LIN {X 0,Y 256.443,Z 273.526,A -85,B 0,C 180,E1 -18716.858,E2 -18716.858} C_VEL
LIN {X 0,Y 256.695,Z 273.51,A -85,B 0,C 180,E1 -18718.431,E2 -18718.431} C_VEL
LIN {X 0,Y 256.584,Z 273.506,A -85,B 0,C 180,E1 -18722.128,E2 -18722.128} C_VEL
LIN {X 0,Y 255.761,Z 273.619,A -85,B 0,C 180,E1 -18723.437,E2 -18723.437} C_VEL
LIN {X 0,Y 252.839,Z 273.986,A -85,B 0,C 180,E1 -18725.572,E2 -18725.572} C_VEL
LIN {X 0,Y 250.455,Z 274.274,A -85,B 0,C 180,E1 -18727.309,E2 -18727.309} C_VEL
LIN {X 0,Y 249.449,Z 274.4,A -85,B 0,C 180,E1 -18728.656,E2 -18728.656} C_VEL
LIN {X 0,Y 249.37,Z 274.413,A -85,B 0,C 180,E1 -18729.112,E2 -18729.112} C_VEL
LIN {X 0,Y 249.184,Z 274.428,A -85,B 0,C 180,E1 -18733.04,E2 -18733.04} C_VEL
LIN {X 0,Y 249.193,Z 274.444,A -85,B 0,C 180,E1 -18736.486,E2 -18736.486} C_VEL
LIN {X 0,Y 249.077,Z 274.451,A -85,B 0,C 180,E1 -18741.519,E2 -18741.519} C_VEL
LIN {X 0,Y 249.078,Z 274.447,A -85,B 0,C 180,E1 -18745.457,E2 -18745.457} C_VEL
LIN {X 0,Y 249.021,Z 274.443,A -85,B 0,C 180,E1 -18748.968,E2 -18748.968} C_VEL
LIN {X 0,Y 249.023,Z 274.449,A -85,B 0,C 180,E1 -18752.427,E2 -18752.427} C_VEL
LIN {X 0,Y 249.029,Z 274.467,A -85,B 0,C 180,E1 -18756.345,E2 -18756.345} C_VEL
LIN {X 0,Y 248.977,Z 274.467,A -85,B 0,C 180,E1 -18760.484,E2 -18760.484} C_VEL
LIN {X 0,Y 249.005,Z 274.668,A -85,B 0,C 180,E1 -18763.299,E2 -18763.299} C_VEL
LIN {X 0,Y 251.939,Z 284.13,A -85,B 0,C 180,E1 -18767.093,E2 -18767.093} C_VEL
LIN {X 0,Y 254.692,Z 293.785,A -85,B 0,C 180,E1 -18770.605,E2 -18770.605} C_VEL
LIN {X 0,Y 256.851,Z 302.565,A -85,B 0,C 180,E1 -18773.556,E2 -18773.556} C_VEL
LIN {X 0,Y 257.592,Z 305.745,A -85,B 0,C 180,E1 -18774.479,E2 -18774.479} C_VEL
LIN {X 0,Y 262.27,Z 316.515,A -85,B 0,C 180,E1 -18775.675,E2 -18775.675} C_VEL
LIN {X 0,Y 263.173,Z 319.74,A -85,B 0,C 180,E1 -18775.93,E2 -18775.93} C_VEL
LIN {X 0,Y 267.638,Z 349.75,A -85,B 0,C 180,E1 -18777.608,E2 -18777.608} C_VEL
LIN {X 0,Y 270.306,Z 373.324,A -85,B 0,C 180,E1 -18778.747,E2 -18778.747} C_VEL
LIN {X 0,Y 270.85,Z 381.222,A -85,B 0,C 180,E1 -18779.071,E2 -18779.071} C_VEL
LIN {X 0,Y 269.246,Z 418.517,A -85,B 0,C 180,E1 -18780.065,E2 -18780.065} C_VEL
LIN {X 0,Y 267.955,Z 432.124,A -85,B 0,C 180,E1 -18780.704,E2 -18780.704} C_VEL
LIN {X 0,Y 266.124,Z 445.126,A -85,B 0,C 180,E1 -18781.617,E2 -18781.617} C_VEL
LIN {X 0,Y 263.547,Z 457.746,A -85,B 0,C 180,E1 -18782.827,E2 -18782.827} C_VEL
LIN {X 0,Y 260.85,Z 469.017,A -85,B 0,C 180,E1 -18784.25,E2 -18784.25} C_VEL
LIN {X 0,Y 258.114,Z 479.21,A -85,B 0,C 180,E1 -18785.894,E2 -18785.894} C_VEL
LIN {X 0,Y 255.483,Z 488.439,A -85,B 0,C 180,E1 -18787.775,E2 -18787.775} C_VEL
LIN {X 0,Y 252.796,Z 497.481,A -85,B 0,C 180,E1 -18790.089,E2 -18790.089} C_VEL
LIN {X 0,Y 250.941,Z 504.121,A -85,B 0,C 180,E1 -18792.218,E2 -18792.218} C_VEL
LIN {X 0,Y 249.474,Z 509.836,A -85,B 0,C 180,E1 -18794.477,E2 -18794.477} C_VEL
LIN {X 0,Y 248.297,Z 514.754,A -85,B 0,C 180,E1 -18796.912,E2 -18796.912} C_VEL
LIN {X 0,Y 247.635,Z 518.587,A -85,B 0,C 180,E1 -18799.369,E2 -18799.369} C_VEL
LIN {X 0,Y 247.49,Z 521.437,A -85,B 0,C 180,E1 -18801.837,E2 -18801.837} C_VEL
LIN {X 0,Y 247.65,Z 522.833,A -85,B 0,C 180,E1 -18803.481,E2 -18803.481} C_VEL
LIN {X 0,Y 247.793,Z 523.809,A -85,B 0,C 180,E1 -18805.118,E2 -18805.118} C_VEL
LIN {X 0,Y 248.089,Z 524.353,A -85,B 0,C 180,E1 -18806.751,E2 -18806.751} C_VEL
LIN {X 0,Y 248.279,Z 524.479,A -85,B 0,C 180,E1 -18808.377,E2 -18808.377} C_VEL
LIN {X 0,Y 248.404,Z 524.194,A -85,B 0,C 180,E1 -18809.999,E2 -18809.999} C_VEL
LIN {X 0,Y 248.339,Z 523.474,A -85,B 0,C 180,E1 -18811.621,E2 -18811.621} C_VEL
LIN {X 0,Y 248.24,Z 522.282,A -85,B 0,C 180,E1 -18813.245,E2 -18813.245} C_VEL
LIN {X 0,Y 247.888,Z 519.656,A -85,B 0,C 180,E1 -18815.694,E2 -18815.694} C_VEL
LIN {X 0,Y 247.682,Z 515.965,A -85,B 0,C 180,E1 -18818.156,E2 -18818.156} C_VEL
LIN {X 0,Y 247.779,Z 511.131,A -85,B 0,C 180,E1 -18820.623,E2 -18820.623} C_VEL
LIN {X 0,Y 248.462,Z 503.88,A -85,B 0,C 180,E1 -18823.494,E2 -18823.494} C_VEL
LIN {X 0,Y 249.454,Z 496.031,A -85,B 0,C 180,E1 -18825.943,E2 -18825.943} C_VEL
LIN {X 0,Y 250.831,Z 488.044,A -85,B 0,C 180,E1 -18827.95,E2 -18827.95} C_VEL
LIN {X 0,Y 252.264,Z 479.373,A -85,B 0,C 180,E1 -18829.742,E2 -18829.742} C_VEL
LIN {X 0,Y 254.056,Z 468.801,A -85,B 0,C 180,E1 -18831.501,E2 -18831.501} C_VEL
LIN {X 0,Y 255.949,Z 457.085,A -85,B 0,C 180,E1 -18833.033,E2 -18833.033} C_VEL
LIN {X 0,Y 257.624,Z 444.652,A -85,B 0,C 180,E1 -18834.26,E2 -18834.26} C_VEL
LIN {X 0,Y 258.91,Z 431.527,A -85,B 0,C 180,E1 -18835.202,E2 -18835.202} C_VEL
LIN {X 0,Y 259.783,Z 418.703,A -85,B 0,C 180,E1 -18835.809,E2 -18835.809} C_VEL
LIN {X 0,Y 260.834,Z 377.068,A -85,B 0,C 180,E1 -18836.957,E2 -18836.957} C_VEL
LIN {X 0,Y 257.271,Z 335.818,A -85,B 0,C 180,E1 -18838.516,E2 -18838.516} C_VEL
LIN {X 0,Y 254.216,Z 308.569,A -85,B 0,C 180,E1 -18839.693,E2 -18839.693} C_VEL
LIN {X 0,Y 254.746,Z 304.307,A -85,B 0,C 180,E1 -18840.668,E2 -18840.668} C_VEL
LIN {X 0,Y 254.864,Z 300.787,A -85,B 0,C 180,E1 -18841.595,E2 -18841.595} C_VEL
LIN {X 0,Y 252.702,Z 289.84,A -85,B 0,C 180,E1 -18844.757,E2 -18844.757} C_VEL
LIN {X 0,Y 250.099,Z 278.579,A -85,B 0,C 180,E1 -18848.184,E2 -18848.184} C_VEL
LIN {X 0,Y 249.018,Z 274.551,A -85,B 0,C 180,E1 -18849.55,E2 -18849.55} C_VEL
LIN {X 0,Y 248.978,Z 274.464,A -85,B 0,C 180,E1 -18852.785,E2 -18852.785} C_VEL
LIN {X 0,Y 248.973,Z 274.461,A -85,B 0,C 180,E1 -18857.354,E2 -18857.354} C_VEL
LIN {X 0,Y 249.033,Z 274.456,A -85,B 0,C 180,E1 -18862.201,E2 -18862.201} C_VEL
LIN {X 0,Y 249.036,Z 274.459,A -85,B 0,C 180,E1 -18865.638,E2 -18865.638} C_VEL
LIN {X 0,Y 248.987,Z 274.465,A -85,B 0,C 180,E1 -18869.464,E2 -18869.464} C_VEL
LIN {X 0,Y 249.021,Z 274.459,A -85,B 0,C 180,E1 -18873.156,E2 -18873.156} C_VEL
LIN {X 0,Y 249.043,Z 274.459,A -85,B 0,C 180,E1 -18876.729,E2 -18876.729} C_VEL
LIN {X 0,Y 249.039,Z 274.46,A -85,B 0,C 180,E1 -18880.206,E2 -18880.206} C_VEL
LIN {X 0,Y 249.149,Z 274.443,A -85,B 0,C 180,E1 -18883.616,E2 -18883.616} C_VEL
LIN {X 0,Y 249.224,Z 274.431,A -85,B 0,C 180,E1 -18888.616,E2 -18888.616} C_VEL
LIN {X 0,Y 249.408,Z 274.407,A -85,B 0,C 180,E1 -18891.901,E2 -18891.901} C_VEL
LIN {X 0,Y 249.253,Z 274.436,A -85,B 0,C 180,E1 -18895.148,E2 -18895.148} C_VEL
LIN {X 0,Y 249.648,Z 274.372,A -85,B 0,C 180,E1 -18898.387,E2 -18898.387} C_VEL
LIN {X 0,Y 249.647,Z 274.381,A -85,B 0,C 180,E1 -18901.614,E2 -18901.614} C_VEL
LIN {X 0,Y 249.398,Z 274.408,A -85,B 0,C 180,E1 -18906.665,E2 -18906.665} C_VEL
LIN {X 0,Y 249.324,Z 274.413,A -85,B 0,C 180,E1 -18909.738,E2 -18909.738} C_VEL
LIN {X 0,Y 249.163,Z 274.443,A -85,B 0,C 180,E1 -18914.706,E2 -18914.706} C_VEL
LIN {X 0,Y 249.087,Z 274.44,A -85,B 0,C 180,E1 -18918.082,E2 -18918.082} C_VEL
LIN {X 0,Y 249.036,Z 274.462,A -85,B 0,C 180,E1 -18921.523,E2 -18921.523} C_VEL
LIN {X 0,Y 249.037,Z 274.45,A -85,B 0,C 180,E1 -18925.441,E2 -18925.441} C_VEL
LIN {X 0,Y 249.017,Z 274.464,A -85,B 0,C 180,E1 -18928.969,E2 -18928.969} C_VEL
LIN {X 0,Y 249.02,Z 274.456,A -85,B 0,C 180,E1 -18932.428,E2 -18932.428} C_VEL
LIN {X 0,Y 249.008,Z 274.468,A -85,B 0,C 180,E1 -18936.35,E2 -18936.35} C_VEL
LIN {X 0,Y 248.974,Z 274.454,A -85,B 0,C 180,E1 -18940.485,E2 -18940.485} C_VEL
LIN {X 0,Y 248.958,Z 274.447,A -85,B 0,C 180,E1 -18944.89,E2 -18944.89} C_VEL
LIN {X 0,Y 248.976,Z 274.469,A -85,B 0,C 180,E1 -18947.356,E2 -18947.356} C_VEL
LIN {X 0,Y 249.041,Z 274.433,A -85,B 0,C 180,E1 -18952.202,E2 -18952.202} C_VEL
LIN {X 0,Y 249.041,Z 274.46,A -85,B 0,C 180,E1 -18955.641,E2 -18955.641} C_VEL
LIN {X 0,Y 248.992,Z 274.45,A -85,B 0,C 180,E1 -18959.467,E2 -18959.467} C_VEL
LIN {X 0,Y 249.013,Z 274.466,A -85,B 0,C 180,E1 -18963.157,E2 -18963.157} C_VEL
LIN {X 0,Y 249.007,Z 274.466,A -85,B 0,C 180,E1 -18966.727,E2 -18966.727} C_VEL
LIN {X 0,Y 249.069,Z 274.697,A -85,B 0,C 180,E1 -18968.264,E2 -18968.264} C_VEL
LIN {X 0,Y 249.342,Z 275.779,A -85,B 0,C 180,E1 -18968.528,E2 -18968.528} C_VEL
LIN {X 0,Y 256.786,Z 291.191,A -85,B 0,C 180,E1 -18969.864,E2 -18969.864} C_VEL
LIN {X 0,Y 262.664,Z 305.025,A -85,B 0,C 180,E1 -18970.889,E2 -18970.889} C_VEL
LIN {X 0,Y 261.449,Z 360.767,A -85,B 0,C 180,E1 -18972.438,E2 -18972.438} C_VEL
LIN {X 0,Y 260.873,Z 373.588,A -85,B 0,C 180,E1 -18973.066,E2 -18973.066} C_VEL
LIN {X 0,Y 260.178,Z 386.354,A -85,B 0,C 180,E1 -18974.028,E2 -18974.028} C_VEL
LIN {X 0,Y 258.96,Z 398.602,A -85,B 0,C 180,E1 -18975.261,E2 -18975.261} C_VEL
LIN {X 0,Y 257.48,Z 410.104,A -85,B 0,C 180,E1 -18976.786,E2 -18976.786} C_VEL
LIN {X 0,Y 256.054,Z 420.419,A -85,B 0,C 180,E1 -18978.523,E2 -18978.523} C_VEL
LIN {X 0,Y 254.596,Z 429.735,A -85,B 0,C 180,E1 -18980.467,E2 -18980.467} C_VEL
LIN {X 0,Y 252.927,Z 438.733,A -85,B 0,C 180,E1 -18982.818,E2 -18982.818} C_VEL
LIN {X 0,Y 251.555,Z 445.985,A -85,B 0,C 180,E1 -18985.193,E2 -18985.193} C_VEL
LIN {X 0,Y 250.513,Z 451.8,A -85,B 0,C 180,E1 -18987.589,E2 -18987.589} C_VEL
LIN {X 0,Y 249.731,Z 456.398,A -85,B 0,C 180,E1 -18990.001,E2 -18990.001} C_VEL
LIN {X 0,Y 249.118,Z 459.929,A -85,B 0,C 180,E1 -18992.426,E2 -18992.426} C_VEL
LIN {X 0,Y 248.925,Z 462.45,A -85,B 0,C 180,E1 -18994.859,E2 -18994.859} C_VEL
LIN {X 0,Y 248.891,Z 463.645,A -85,B 0,C 180,E1 -18996.486,E2 -18996.486} C_VEL
LIN {X 0,Y 249.017,Z 464.801,A -85,B 0,C 180,E1 -18999.75,E2 -18999.75} C_VEL
LIN {X 0,Y 249.606,Z 464.433,A -85,B 0,C 180,E1 -19003.018,E2 -19003.018} C_VEL
LIN {X 0,Y 250.697,Z 462.408,A -85,B 0,C 180,E1 -19006.281,E2 -19006.281} C_VEL
LIN {X 0,Y 251.679,Z 460.33,A -85,B 0,C 180,E1 -19008.297,E2 -19008.297} C_VEL
LIN {X 0,Y 253.326,Z 456.162,A -85,B 0,C 180,E1 -19011.141,E2 -19011.141} C_VEL
LIN {X 0,Y 255.106,Z 451.378,A -85,B 0,C 180,E1 -19013.545,E2 -19013.545} C_VEL
LIN {X 0,Y 257.245,Z 445.293,A -85,B 0,C 180,E1 -19015.921,E2 -19015.921} C_VEL
LIN {X 0,Y 259.642,Z 437.642,A -85,B 0,C 180,E1 -19018.274,E2 -19018.274} C_VEL
LIN {X 0,Y 261.926,Z 429.739,A -85,B 0,C 180,E1 -19020.205,E2 -19020.205} C_VEL
LIN {X 0,Y 264.26,Z 420.034,A -85,B 0,C 180,E1 -19022.134,E2 -19022.134} C_VEL
LIN {X 0,Y 266.613,Z 409.146,A -85,B 0,C 180,E1 -19023.839,E2 -19023.839} C_VEL
LIN {X 0,Y 268.486,Z 398.379,A -85,B 0,C 180,E1 -19025.161,E2 -19025.161} C_VEL
LIN {X 0,Y 269.94,Z 387.778,A -85,B 0,C 180,E1 -19026.186,E2 -19026.186} C_VEL
LIN {X 0,Y 271.093,Z 375.462,A -85,B 0,C 180,E1 -19027.088,E2 -19027.088} C_VEL
LIN {X 0,Y 271.773,Z 363.252,A -85,B 0,C 180,E1 -19027.707,E2 -19027.707} C_VEL
LIN {X 0,Y 272.781,Z 328.656,A -85,B 0,C 180,E1 -19028.694,E2 -19028.694} C_VEL
LIN {X 0,Y 273.176,Z 316.973,A -85,B 0,C 180,E1 -19029.004,E2 -19029.004} C_VEL
LIN {X 0,Y 265.765,Z 302.535,A -85,B 0,C 180,E1 -19030.616,E2 -19030.616} C_VEL
LIN {X 0,Y 258.181,Z 289.71,A -85,B 0,C 180,E1 -19032.334,E2 -19032.334} C_VEL
LIN {X 0,Y 253.23,Z 282.015,A -85,B 0,C 180,E1 -19033.51,E2 -19033.51} C_VEL
LIN {X 0,Y 251.177,Z 278.766,A -85,B 0,C 180,E1 -19034.02,E2 -19034.02} C_VEL
LIN {X 0,Y 249.479,Z 276.328,A -85,B 0,C 180,E1 -19034.45,E2 -19034.45} C_VEL
LIN {X 0,Y 249.065,Z 275,A -85,B 0,C 180,E1 -19034.691,E2 -19034.691} C_VEL
LIN {X 0,Y 248.967,Z 274.504,A -85,B 0,C 180,E1 -19035.112,E2 -19035.112} C_VEL
LIN {X 0,Y 248.979,Z 274.473,A -85,B 0,C 180,E1 -19039.516,E2 -19039.516} C_VEL
LIN {X 0,Y 249.012,Z 274.438,A -85,B 0,C 180,E1 -19043.651,E2 -19043.651} C_VEL
LIN {X 0,Y 249.03,Z 274.435,A -85,B 0,C 180,E1 -19047.848,E2 -19047.848} C_VEL
LIN {X 0,Y 249.038,Z 274.432,A -85,B 0,C 180,E1 -19051.33,E2 -19051.33} C_VEL
LIN {X 0,Y 249.1,Z 274.444,A -85,B 0,C 180,E1 -19054.962,E2 -19054.962} C_VEL
LIN {X 0,Y 249.089,Z 274.4,A -85,B 0,C 180,E1 -19058.604,E2 -19058.604} C_VEL
LIN {X 0,Y 249.241,Z 274.436,A -85,B 0,C 180,E1 -19063.621,E2 -19063.621} C_VEL
LIN {X 0,Y 249.24,Z 274.437,A -85,B 0,C 180,E1 -19068.616,E2 -19068.616} C_VEL
LIN {X 0,Y 249.414,Z 274.405,A -85,B 0,C 180,E1 -19071.9,E2 -19071.9} C_VEL
LIN {X 0,Y 249.253,Z 274.424,A -85,B 0,C 180,E1 -19075.147,E2 -19075.147} C_VEL
LIN {X 0,Y 249.655,Z 274.387,A -85,B 0,C 180,E1 -19078.386,E2 -19078.386} C_VEL
LIN {X 0,Y 249.561,Z 274.381,A -85,B 0,C 180,E1 -19082.058,E2 -19082.058} C_VEL
LIN {X 0,Y 249.421,Z 274.403,A -85,B 0,C 180,E1 -19086.471,E2 -19086.471} C_VEL
LIN {X 0,Y 249.37,Z 274.413,A -85,B 0,C 180,E1 -19089.112,E2 -19089.112} C_VEL
LIN {X 0,Y 248.682,Z 274.51,A -85,B 0,C 180,E1 -19090.458,E2 -19090.458} C_VEL
LIN {X 0,Y 245.733,Z 274.877,A -85,B 0,C 180,E1 -19092.65,E2 -19092.65} C_VEL
LIN {X 0,Y 243.238,Z 275.182,A -85,B 0,C 180,E1 -19094.436,E2 -19094.436} C_VEL
LIN {X 0,Y 242.186,Z 275.318,A -85,B 0,C 180,E1 -19095.824,E2 -19095.824} C_VEL
LIN {X 0,Y 242.111,Z 275.322,A -85,B 0,C 180,E1 -19096.295,E2 -19096.295} C_VEL
LIN {X 0,Y 242.021,Z 275.339,A -85,B 0,C 180,E1 -19100.393,E2 -19100.393} C_VEL
LIN {X 0,Y 242.021,Z 275.34,A -85,B 0,C 180,E1 -19103.988,E2 -19103.988} C_VEL
LIN {X 0,Y 241.953,Z 275.313,A -85,B 0,C 180,E1 -19107.694,E2 -19107.694} C_VEL
LIN {X 0,Y 241.946,Z 275.344,A -85,B 0,C 180,E1 -19111.524,E2 -19111.524} C_VEL
LIN {X 0,Y 242.004,Z 275.33,A -85,B 0,C 180,E1 -19115.597,E2 -19115.597} C_VEL
LIN {X 0,Y 241.938,Z 275.334,A -85,B 0,C 180,E1 -19119.722,E2 -19119.722} C_VEL
LIN {X 0,Y 241.957,Z 275.593,A -85,B 0,C 180,E1 -19122.09,E2 -19122.09} C_VEL
LIN {X 0,Y 244.787,Z 284.528,A -85,B 0,C 180,E1 -19125.87,E2 -19125.87} C_VEL
LIN {X 0,Y 247.628,Z 294.176,A -85,B 0,C 180,E1 -19129.57,E2 -19129.57} C_VEL
LIN {X 0,Y 250.128,Z 304.192,A -85,B 0,C 180,E1 -19133.037,E2 -19133.037} C_VEL
LIN {X 0,Y 254.27,Z 313.334,A -85,B 0,C 180,E1 -19134.196,E2 -19134.196} C_VEL
LIN {X 0,Y 257.472,Z 320.978,A -85,B 0,C 180,E1 -19135.025,E2 -19135.025} C_VEL
LIN {X 0,Y 261.882,Z 351.317,A -85,B 0,C 180,E1 -19136.777,E2 -19136.777} C_VEL
LIN {X 0,Y 264.447,Z 374.596,A -85,B 0,C 180,E1 -19137.935,E2 -19137.935} C_VEL
LIN {X 0,Y 264.899,Z 382.546,A -85,B 0,C 180,E1 -19138.26,E2 -19138.26} C_VEL
LIN {X 0,Y 263.417,Z 416.986,A -85,B 0,C 180,E1 -19139.194,E2 -19139.194} C_VEL
LIN {X 0,Y 262.11,Z 430.421,A -85,B 0,C 180,E1 -19139.818,E2 -19139.818} C_VEL
LIN {X 0,Y 260.286,Z 443.122,A -85,B 0,C 180,E1 -19140.699,E2 -19140.699} C_VEL
LIN {X 0,Y 258.002,Z 454.457,A -85,B 0,C 180,E1 -19141.751,E2 -19141.751} C_VEL
LIN {X 0,Y 255.108,Z 466.171,A -85,B 0,C 180,E1 -19143.185,E2 -19143.185} C_VEL
LIN {X 0,Y 252.217,Z 476.733,A -85,B 0,C 180,E1 -19144.853,E2 -19144.853} C_VEL
LIN {X 0,Y 249.424,Z 486.3,A -85,B 0,C 180,E1 -19146.767,E2 -19146.767} C_VEL
LIN {X 0,Y 246.544,Z 495.562,A -85,B 0,C 180,E1 -19149.125,E2 -19149.125} C_VEL
LIN {X 0,Y 244.287,Z 503.086,A -85,B 0,C 180,E1 -19151.551,E2 -19151.551} C_VEL
LIN {X 0,Y 242.606,Z 509.188,A -85,B 0,C 180,E1 -19154.025,E2 -19154.025} C_VEL
LIN {X 0,Y 241.348,Z 514.06,A -85,B 0,C 180,E1 -19156.528,E2 -19156.528} C_VEL
LIN {X 0,Y 240.602,Z 517.848,A -85,B 0,C 180,E1 -19159.055,E2 -19159.055} C_VEL
LIN {X 0,Y 240.403,Z 520.657,A -85,B 0,C 180,E1 -19161.594,E2 -19161.594} C_VEL
LIN {X 0,Y 240.57,Z 522.085,A -85,B 0,C 180,E1 -19163.352,E2 -19163.352} C_VEL
LIN {X 0,Y 241.011,Z 523.508,A -85,B 0,C 180,E1 -19166.656,E2 -19166.656} C_VEL
LIN {X 0,Y 241.227,Z 523.62,A -85,B 0,C 180,E1 -19168.33,E2 -19168.33} C_VEL
LIN {X 0,Y 241.355,Z 523.318,A -85,B 0,C 180,E1 -19169.999,E2 -19169.999} C_VEL
LIN {X 0,Y 241.29,Z 522.569,A -85,B 0,C 180,E1 -19171.668,E2 -19171.668} C_VEL
LIN {X 0,Y 241.157,Z 521.345,A -85,B 0,C 180,E1 -19173.341,E2 -19173.341} C_VEL
LIN {X 0,Y 240.816,Z 518.678,A -85,B 0,C 180,E1 -19175.862,E2 -19175.862} C_VEL
LIN {X 0,Y 240.605,Z 514.94,A -85,B 0,C 180,E1 -19178.397,E2 -19178.397} C_VEL
LIN {X 0,Y 240.75,Z 510.06,A -85,B 0,C 180,E1 -19180.937,E2 -19180.937} C_VEL
LIN {X 0,Y 241.494,Z 502.756,A -85,B 0,C 180,E1 -19183.891,E2 -19183.891} C_VEL
LIN {X 0,Y 242.52,Z 494.817,A -85,B 0,C 180,E1 -19186.411,E2 -19186.411} C_VEL
LIN {X 0,Y 243.992,Z 486.755,A -85,B 0,C 180,E1 -19188.471,E2 -19188.471} C_VEL
LIN {X 0,Y 245.779,Z 476.927,A -85,B 0,C 180,E1 -19190.504,E2 -19190.504} C_VEL
LIN {X 0,Y 247.572,Z 466.003,A -85,B 0,C 180,E1 -19192.313,E2 -19192.313} C_VEL
LIN {X 0,Y 249.139,Z 457.076,A -85,B 0,C 180,E1 -19193.48,E2 -19193.48} C_VEL
LIN {X 0,Y 250.862,Z 444.998,A -85,B 0,C 180,E1 -19194.737,E2 -19194.737} C_VEL
LIN {X 0,Y 252.189,Z 432.293,A -85,B 0,C 180,E1 -19195.701,E2 -19195.701} C_VEL
LIN {X 0,Y 253.157,Z 419.171,A -85,B 0,C 180,E1 -19196.37,E2 -19196.37} C_VEL
LIN {X 0,Y 254.296,Z 377.496,A -85,B 0,C 180,E1 -19197.563,E2 -19197.563} C_VEL
LIN {X 0,Y 250.733,Z 335.752,A -85,B 0,C 180,E1 -19199.195,E2 -19199.195} C_VEL
LIN {X 0,Y 247.598,Z 307.785,A -85,B 0,C 180,E1 -19200.449,E2 -19200.449} C_VEL
LIN {X 0,Y 247.883,Z 305.078,A -85,B 0,C 180,E1 -19201.028,E2 -19201.028} C_VEL
LIN {X 0,Y 247.794,Z 301.329,A -85,B 0,C 180,E1 -19202.064,E2 -19202.064} C_VEL
LIN {X 0,Y 245.385,Z 289.262,A -85,B 0,C 180,E1 -19205.681,E2 -19205.681} C_VEL
LIN {X 0,Y 243.108,Z 279.773,A -85,B 0,C 180,E1 -19208.69,E2 -19208.69} C_VEL
LIN {X 0,Y 241.969,Z 275.448,A -85,B 0,C 180,E1 -19210.189,E2 -19210.189} C_VEL
LIN {X 0,Y 241.894,Z 275.323,A -85,B 0,C 180,E1 -19214.208,E2 -19214.208} C_VEL
LIN {X 0,Y 241.902,Z 275.351,A -85,B 0,C 180,E1 -19218.07,E2 -19218.07} C_VEL
LIN {X 0,Y 241.978,Z 275.335,A -85,B 0,C 180,E1 -19222.416,E2 -19222.416} C_VEL
LIN {X 0,Y 241.971,Z 275.333,A -85,B 0,C 180,E1 -19226.506,E2 -19226.506} C_VEL
LIN {X 0,Y 241.964,Z 275.343,A -85,B 0,C 180,E1 -19230.614,E2 -19230.614} C_VEL
LIN {X 0,Y 242.025,Z 275.326,A -85,B 0,C 180,E1 -19234.178,E2 -19234.178} C_VEL
LIN {X 0,Y 241.984,Z 275.342,A -85,B 0,C 180,E1 -19238.334,E2 -19238.334} C_VEL
LIN {X 0,Y 242.105,Z 275.317,A -85,B 0,C 180,E1 -19243.318,E2 -19243.318} C_VEL
LIN {X 0,Y 242.158,Z 275.315,A -85,B 0,C 180,E1 -19248.279,E2 -19248.279} C_VEL
LIN {X 0,Y 242.362,Z 275.284,A -85,B 0,C 180,E1 -19251.664,E2 -19251.664} C_VEL
LIN {X 0,Y 242.386,Z 275.29,A -85,B 0,C 180,E1 -19253.34,E2 -19253.34} C_VEL
LIN {X 0,Y 242.608,Z 275.248,A -85,B 0,C 180,E1 -19258.34,E2 -19258.34} C_VEL
LIN {X 0,Y 242.606,Z 275.258,A -85,B 0,C 180,E1 -19261.66,E2 -19261.66} C_VEL
LIN {X 0,Y 242.38,Z 275.282,A -85,B 0,C 180,E1 -19266.661,E2 -19266.661} C_VEL
LIN {X 0,Y 242.252,Z 275.294,A -85,B 0,C 180,E1 -19270.025,E2 -19270.025} C_VEL
LIN {X 0,Y 242.113,Z 275.319,A -85,B 0,C 180,E1 -19275.145,E2 -19275.145} C_VEL
LIN {X 0,Y 242.023,Z 275.323,A -85,B 0,C 180,E1 -19278.629,E2 -19278.629} C_VEL
LIN {X 0,Y 241.966,Z 275.345,A -85,B 0,C 180,E1 -19282.185,E2 -19282.185} C_VEL
LIN {X 0,Y 241.98,Z 275.327,A -85,B 0,C 180,E1 -19285.828,E2 -19285.828} C_VEL
LIN {X 0,Y 241.956,Z 275.345,A -85,B 0,C 180,E1 -19289.591,E2 -19289.591} C_VEL
LIN {X 0,Y 241.973,Z 275.33,A -85,B 0,C 180,E1 -19293.494,E2 -19293.494} C_VEL
LIN {X 0,Y 241.979,Z 275.344,A -85,B 0,C 180,E1 -19297.585,E2 -19297.585} C_VEL
LIN {X 0,Y 241.896,Z 275.314,A -85,B 0,C 180,E1 -19301.932,E2 -19301.932} C_VEL
LIN {X 0,Y 241.897,Z 275.347,A -85,B 0,C 180,E1 -19306.582,E2 -19306.582} C_VEL
LIN {X 0,Y 241.991,Z 275.314,A -85,B 0,C 180,E1 -19311.643,E2 -19311.643} C_VEL
LIN {X 0,Y 241.972,Z 275.324,A -85,B 0,C 180,E1 -19314.488,E2 -19314.488} C_VEL
LIN {X 0,Y 241.947,Z 275.334,A -85,B 0,C 180,E1 -19318.477,E2 -19318.477} C_VEL
LIN {X 0,Y 241.951,Z 275.348,A -85,B 0,C 180,E1 -19322.307,E2 -19322.307} C_VEL
LIN {X 0,Y 241.958,Z 275.334,A -85,B 0,C 180,E1 -19326.007,E2 -19326.007} C_VEL
LIN {X 0,Y 242.017,Z 275.564,A -85,B 0,C 180,E1 -19327.417,E2 -19327.417} C_VEL
LIN {X 0,Y 242.249,Z 276.524,A -85,B 0,C 180,E1 -19327.687,E2 -19327.687} C_VEL
LIN {X 0,Y 249.041,Z 290.279,A -85,B 0,C 180,E1 -19328.972,E2 -19328.972} C_VEL
LIN {X 0,Y 256.235,Z 306.889,A -85,B 0,C 180,E1 -19330.282,E2 -19330.282} C_VEL
LIN {X 0,Y 254.917,Z 359.495,A -85,B 0,C 180,E1 -19331.757,E2 -19331.757} C_VEL
LIN {X 0,Y 254.428,Z 372.618,A -85,B 0,C 180,E1 -19332.364,E2 -19332.364} C_VEL
LIN {X 0,Y 253.755,Z 385.341,A -85,B 0,C 180,E1 -19333.302,E2 -19333.302} C_VEL
LIN {X 0,Y 252.608,Z 397.143,A -85,B 0,C 180,E1 -19334.469,E2 -19334.469} C_VEL
LIN {X 0,Y 251.207,Z 407.876,A -85,B 0,C 180,E1 -19335.831,E2 -19335.831} C_VEL
LIN {X 0,Y 249.657,Z 418.811,A -85,B 0,C 180,E1 -19337.606,E2 -19337.606} C_VEL
LIN {X 0,Y 247.989,Z 429.41,A -85,B 0,C 180,E1 -19339.799,E2 -19339.799} C_VEL
LIN {X 0,Y 246.504,Z 437.274,A -85,B 0,C 180,E1 -19341.805,E2 -19341.805} C_VEL
LIN {X 0,Y 244.969,Z 444.994,A -85,B 0,C 180,E1 -19344.238,E2 -19344.238} C_VEL
LIN {X 0,Y 243.856,Z 451.146,A -85,B 0,C 180,E1 -19346.696,E2 -19346.696} C_VEL
LIN {X 0,Y 242.943,Z 456.062,A -85,B 0,C 180,E1 -19349.172,E2 -19349.172} C_VEL
LIN {X 0,Y 242.213,Z 459.89,A -85,B 0,C 180,E1 -19351.663,E2 -19351.663} C_VEL
LIN {X 0,Y 241.908,Z 461.867,A -85,B 0,C 180,E1 -19353.332,E2 -19353.332} C_VEL
LIN {X 0,Y 241.884,Z 463.418,A -85,B 0,C 180,E1 -19355.001,E2 -19355.001} C_VEL
LIN {X 0,Y 241.852,Z 464.567,A -85,B 0,C 180,E1 -19356.675,E2 -19356.675} C_VEL
LIN {X 0,Y 242.002,Z 465.669,A -85,B 0,C 180,E1 -19360.035,E2 -19360.035} C_VEL
LIN {X 0,Y 242.28,Z 465.653,A -85,B 0,C 180,E1 -19361.716,E2 -19361.716} C_VEL
LIN {X 0,Y 242.663,Z 465.226,A -85,B 0,C 180,E1 -19363.397,E2 -19363.397} C_VEL
LIN {X 0,Y 243.859,Z 463.144,A -85,B 0,C 180,E1 -19366.751,E2 -19366.751} C_VEL
LIN {X 0,Y 244.837,Z 461.174,A -85,B 0,C 180,E1 -19368.689,E2 -19368.689} C_VEL
LIN {X 0,Y 246.656,Z 456.785,A -85,B 0,C 180,E1 -19371.741,E2 -19371.741} C_VEL
LIN {X 0,Y 248.541,Z 451.938,A -85,B 0,C 180,E1 -19374.206,E2 -19374.206} C_VEL
LIN {X 0,Y 250.802,Z 445.782,A -85,B 0,C 180,E1 -19376.638,E2 -19376.638} C_VEL
LIN {X 0,Y 253.334,Z 438.007,A -85,B 0,C 180,E1 -19379.044,E2 -19379.044} C_VEL
LIN {X 0,Y 255.728,Z 430.005,A -85,B 0,C 180,E1 -19381.017,E2 -19381.017} C_VEL
LIN {X 0,Y 258.215,Z 420.182,A -85,B 0,C 180,E1 -19382.98,E2 -19382.98} C_VEL
LIN {X 0,Y 260.385,Z 410.46,A -85,B 0,C 180,E1 -19384.528,E2 -19384.528} C_VEL
LIN {X 0,Y 262.34,Z 399.847,A -85,B 0,C 180,E1 -19385.875,E2 -19385.875} C_VEL
LIN {X 0,Y 264.002,Z 388.423,A -85,B 0,C 180,E1 -19386.999,E2 -19386.999} C_VEL
LIN {X 0,Y 265.177,Z 376.226,A -85,B 0,C 180,E1 -19387.91,E2 -19387.91} C_VEL
LIN {X 0,Y 265.889,Z 364.161,A -85,B 0,C 180,E1 -19388.532,E2 -19388.532} C_VEL
LIN {X 0,Y 266.802,Z 334.001,A -85,B 0,C 180,E1 -19389.42,E2 -19389.42} C_VEL
LIN {X 0,Y 267.243,Z 319.117,A -85,B 0,C 180,E1 -19389.836,E2 -19389.836} C_VEL
LIN {X 0,Y 260.244,Z 305.541,A -85,B 0,C 180,E1 -19391.429,E2 -19391.429} C_VEL
LIN {X 0,Y 252.923,Z 293.235,A -85,B 0,C 180,E1 -19393.161,E2 -19393.161} C_VEL
LIN {X 0,Y 246.996,Z 283.882,A -85,B 0,C 180,E1 -19394.654,E2 -19394.654} C_VEL
LIN {X 0,Y 244.783,Z 280.43,A -85,B 0,C 180,E1 -19395.238,E2 -19395.238} C_VEL
LIN {X 0,Y 242.596,Z 277.69,A -85,B 0,C 180,E1 -19395.805,E2 -19395.805} C_VEL
LIN {X 0,Y 241.966,Z 275.822,A -85,B 0,C 180,E1 -19396.155,E2 -19396.155} C_VEL
LIN {X 0,Y 241.9,Z 275.38,A -85,B 0,C 180,E1 -19396.579,E2 -19396.579} C_VEL
LIN {X 0,Y 241.993,Z 275.309,A -85,B 0,C 180,E1 -19401.64,E2 -19401.64} C_VEL
LIN {X 0,Y 241.973,Z 275.326,A -85,B 0,C 180,E1 -19404.486,E2 -19404.486} C_VEL
LIN {X 0,Y 241.947,Z 275.307,A -85,B 0,C 180,E1 -19408.475,E2 -19408.475} C_VEL
LIN {X 0,Y 241.96,Z 275.332,A -85,B 0,C 180,E1 -19412.306,E2 -19412.306} C_VEL
LIN {X 0,Y 242.023,Z 275.3,A -85,B 0,C 180,E1 -19416.012,E2 -19416.012} C_VEL
LIN {X 0,Y 242.027,Z 275.287,A -85,B 0,C 180,E1 -19419.607,E2 -19419.607} C_VEL
LIN {X 0,Y 242.162,Z 275.321,A -85,B 0,C 180,E1 -19423.278,E2 -19423.278} C_VEL
LIN {X 0,Y 242.177,Z 275.318,A -85,B 0,C 180,E1 -19428.279,E2 -19428.279} C_VEL
LIN {X 0,Y 242.368,Z 275.28,A -85,B 0,C 180,E1 -19431.663,E2 -19431.663} C_VEL
LIN {X 0,Y 242.392,Z 275.291,A -85,B 0,C 180,E1 -19433.34,E2 -19433.34} C_VEL
LIN {X 0,Y 242.615,Z 275.263,A -85,B 0,C 180,E1 -19438.34,E2 -19438.34} C_VEL
LIN {X 0,Y 242.614,Z 275.245,A -85,B 0,C 180,E1 -19441.66,E2 -19441.66} C_VEL
LIN {X 0,Y 242.392,Z 275.276,A -85,B 0,C 180,E1 -19446.66,E2 -19446.66} C_VEL
LIN {X 0,Y 242.259,Z 275.309,A -85,B 0,C 180,E1 -19450.024,E2 -19450.024} C_VEL
LIN {X 0,Y 242.136,Z 275.321,A -85,B 0,C 180,E1 -19455.142,E2 -19455.142} C_VEL
LIN {X 0,Y 242.111,Z 275.322,A -85,B 0,C 180,E1 -19456.295,E2 -19456.295} C_VEL
LIN {X 0,Y 241.455,Z 275.408,A -85,B 0,C 180,E1 -19457.683,E2 -19457.683} C_VEL
LIN {X 0,Y 238.55,Z 275.772,A -85,B 0,C 180,E1 -19459.946,E2 -19459.946} C_VEL
LIN {X 0,Y 236.065,Z 276.075,A -85,B 0,C 180,E1 -19461.79,E2 -19461.79} C_VEL
LIN {X 0,Y 235,Z 276.209,A -85,B 0,C 180,E1 -19463.223,E2 -19463.223} C_VEL
LIN {X 0,Y 234.915,Z 276.215,A -85,B 0,C 180,E1 -19463.709,E2 -19463.709} C_VEL
LIN {X 0,Y 234.939,Z 276.19,A -85,B 0,C 180,E1 -19466.661,E2 -19466.661} C_VEL
LIN {X 0,Y 234.892,Z 276.227,A -85,B 0,C 180,E1 -19470.573,E2 -19470.573} C_VEL
LIN {X 0,Y 234.924,Z 276.199,A -85,B 0,C 180,E1 -19474.639,E2 -19474.639} C_VEL
LIN {X 0,Y 234.91,Z 276.205,A -85,B 0,C 180,E1 -19478.935,E2 -19478.935} C_VEL
LIN {X 0,Y 234.901,Z 276.439,A -85,B 0,C 180,E1 -19480.738,E2 -19480.738} C_VEL
LIN {X 0,Y 237.841,Z 285.593,A -85,B 0,C 180,E1 -19484.832,E2 -19484.832} C_VEL
LIN {X 0,Y 240.727,Z 295.335,A -85,B 0,C 180,E1 -19488.743,E2 -19488.743} C_VEL
LIN {X 0,Y 242.784,Z 303.231,A -85,B 0,C 180,E1 -19491.576,E2 -19491.576} C_VEL
LIN {X 0,Y 248.608,Z 315.63,A -85,B 0,C 180,E1 -19493.235,E2 -19493.235} C_VEL
LIN {X 0,Y 252.102,Z 323.853,A -85,B 0,C 180,E1 -19494.181,E2 -19494.181} C_VEL
LIN {X 0,Y 256.191,Z 352.847,A -85,B 0,C 180,E1 -19495.907,E2 -19495.907} C_VEL
LIN {X 0,Y 258.754,Z 377.1,A -85,B 0,C 180,E1 -19497.145,E2 -19497.145} C_VEL
LIN {X 0,Y 259.019,Z 383.917,A -85,B 0,C 180,E1 -19497.414,E2 -19497.414} C_VEL
LIN {X 0,Y 257.503,Z 417.008,A -85,B 0,C 180,E1 -19498.34,E2 -19498.34} C_VEL
LIN {X 0,Y 256.107,Z 430.27,A -85,B 0,C 180,E1 -19498.977,E2 -19498.977} C_VEL
LIN {X 0,Y 254.133,Z 443.307,A -85,B 0,C 180,E1 -19499.918,E2 -19499.918} C_VEL
LIN {X 0,Y 251.372,Z 455.943,A -85,B 0,C 180,E1 -19501.165,E2 -19501.165} C_VEL
LIN {X 0,Y 248.446,Z 467.223,A -85,B 0,C 180,E1 -19502.634,E2 -19502.634} C_VEL
LIN {X 0,Y 245.488,Z 477.426,A -85,B 0,C 180,E1 -19504.341,E2 -19504.341} C_VEL
LIN {X 0,Y 242.357,Z 487.484,A -85,B 0,C 180,E1 -19506.501,E2 -19506.501} C_VEL
LIN {X 0,Y 239.438,Z 496.397,A -85,B 0,C 180,E1 -19508.926,E2 -19508.926} C_VEL
LIN {X 0,Y 237.026,Z 504.008,A -85,B 0,C 180,E1 -19511.591,E2 -19511.591} C_VEL
LIN {X 0,Y 235.196,Z 510.252,A -85,B 0,C 180,E1 -19514.399,E2 -19514.399} C_VEL
LIN {X 0,Y 234.06,Z 514.71,A -85,B 0,C 180,E1 -19516.985,E2 -19516.985} C_VEL
LIN {X 0,Y 233.443,Z 518.13,A -85,B 0,C 180,E1 -19519.593,E2 -19519.593} C_VEL
LIN {X 0,Y 233.463,Z 521.241,A -85,B 0,C 180,E1 -19523.083,E2 -19523.083} C_VEL
LIN {X 0,Y 233.62,Z 522.152,A -85,B 0,C 180,E1 -19524.821,E2 -19524.821} C_VEL
LIN {X 0,Y 233.933,Z 522.662,A -85,B 0,C 180,E1 -19526.555,E2 -19526.555} C_VEL
LIN {X 0,Y 234.175,Z 522.761,A -85,B 0,C 180,E1 -19528.28,E2 -19528.28} C_VEL
LIN {X 0,Y 234.305,Z 522.441,A -85,B 0,C 180,E1 -19529.999,E2 -19529.999} C_VEL
LIN {X 0,Y 234.239,Z 521.656,A -85,B 0,C 180,E1 -19531.719,E2 -19531.719} C_VEL
LIN {X 0,Y 234.076,Z 520.406,A -85,B 0,C 180,E1 -19533.442,E2 -19533.442} C_VEL
LIN {X 0,Y 233.737,Z 517.696,A -85,B 0,C 180,E1 -19536.04,E2 -19536.04} C_VEL
LIN {X 0,Y 233.522,Z 513.909,A -85,B 0,C 180,E1 -19538.654,E2 -19538.654} C_VEL
LIN {X 0,Y 233.734,Z 508.986,A -85,B 0,C 180,E1 -19541.27,E2 -19541.27} C_VEL
LIN {X 0,Y 234.396,Z 502.782,A -85,B 0,C 180,E1 -19543.878,E2 -19543.878} C_VEL
LIN {X 0,Y 235.424,Z 495.062,A -85,B 0,C 180,E1 -19546.474,E2 -19546.474} C_VEL
LIN {X 0,Y 237.024,Z 486.538,A -85,B 0,C 180,E1 -19548.771,E2 -19548.771} C_VEL
LIN {X 0,Y 238.71,Z 477.738,A -85,B 0,C 180,E1 -19550.688,E2 -19550.688} C_VEL
LIN {X 0,Y 240.335,Z 468.472,A -85,B 0,C 180,E1 -19552.342,E2 -19552.342} C_VEL
LIN {X 0,Y 242.333,Z 457.064,A -85,B 0,C 180,E1 -19553.954,E2 -19553.954} C_VEL
LIN {X 0,Y 244.124,Z 445.242,A -85,B 0,C 180,E1 -19555.24,E2 -19555.24} C_VEL
LIN {X 0,Y 245.546,Z 432.285,A -85,B 0,C 180,E1 -19556.278,E2 -19556.278} C_VEL
LIN {X 0,Y 246.567,Z 419.589,A -85,B 0,C 180,E1 -19556.959,E2 -19556.959} C_VEL
LIN {X 0,Y 247.327,Z 397.306,A -85,B 0,C 180,E1 -19557.649,E2 -19557.649} C_VEL
LIN {X 0,Y 247.741,Z 377.651,A -85,B 0,C 180,E1 -19558.214,E2 -19558.214} C_VEL
LIN {X 0,Y 244.416,Z 337.54,A -85,B 0,C 180,E1 -19559.83,E2 -19559.83} C_VEL
LIN {X 0,Y 241.001,Z 306.9,A -85,B 0,C 180,E1 -19561.248,E2 -19561.248} C_VEL
LIN {X 0,Y 241.111,Z 303.98,A -85,B 0,C 180,E1 -19561.928,E2 -19561.928} C_VEL
LIN {X 0,Y 239.024,Z 293.187,A -85,B 0,C 180,E1 -19565.236,E2 -19565.236} C_VEL
LIN {X 0,Y 236.652,Z 282.87,A -85,B 0,C 180,E1 -19568.581,E2 -19568.581} C_VEL
LIN {X 0,Y 234.893,Z 276.337,A -85,B 0,C 180,E1 -19570.896,E2 -19570.896} C_VEL
LIN {X 0,Y 234.861,Z 276.198,A -85,B 0,C 180,E1 -19574.096,E2 -19574.096} C_VEL
LIN {X 0,Y 234.848,Z 276.232,A -85,B 0,C 180,E1 -19578.825,E2 -19578.825} C_VEL
LIN {X 0,Y 234.912,Z 276.213,A -85,B 0,C 180,E1 -19581.078,E2 -19581.078} C_VEL
LIN {X 0,Y 234.921,Z 276.219,A -85,B 0,C 180,E1 -19585.361,E2 -19585.361} C_VEL
LIN {X 0,Y 234.887,Z 276.219,A -85,B 0,C 180,E1 -19589.426,E2 -19589.426} C_VEL
LIN {X 0,Y 234.961,Z 276.207,A -85,B 0,C 180,E1 -19593.806,E2 -19593.806} C_VEL
LIN {X 0,Y 234.957,Z 276.217,A -85,B 0,C 180,E1 -19598.008,E2 -19598.008} C_VEL
LIN {X 0,Y 235.047,Z 276.193,A -85,B 0,C 180,E1 -19603.093,E2 -19603.093} C_VEL
LIN {X 0,Y 235.09,Z 276.197,A -85,B 0,C 180,E1 -19607.921,E2 -19607.921} C_VEL
LIN {X 0,Y 235.302,Z 276.161,A -85,B 0,C 180,E1 -19611.412,E2 -19611.412} C_VEL
LIN {X 0,Y 235.337,Z 276.169,A -85,B 0,C 180,E1 -19613.14,E2 -19613.14} C_VEL
LIN {X 0,Y 235.567,Z 276.124,A -85,B 0,C 180,E1 -19618.291,E2 -19618.291} C_VEL
LIN {X 0,Y 235.565,Z 276.135,A -85,B 0,C 180,E1 -19621.71,E2 -19621.71} C_VEL
LIN {X 0,Y 235.331,Z 276.158,A -85,B 0,C 180,E1 -19626.861,E2 -19626.861} C_VEL
LIN {X 0,Y 235.177,Z 276.177,A -85,B 0,C 180,E1 -19630.33,E2 -19630.33} C_VEL
LIN {X 0,Y 235.063,Z 276.196,A -85,B 0,C 180,E1 -19635.61,E2 -19635.61} C_VEL
LIN {X 0,Y 234.962,Z 276.207,A -85,B 0,C 180,E1 -19639.21,E2 -19639.21} C_VEL
LIN {X 0,Y 234.91,Z 276.22,A -85,B 0,C 180,E1 -19642.889,E2 -19642.889} C_VEL
LIN {X 0,Y 234.898,Z 276.21,A -85,B 0,C 180,E1 -19646.667,E2 -19646.667} C_VEL
LIN {X 0,Y 234.889,Z 276.225,A -85,B 0,C 180,E1 -19650.575,E2 -19650.575} C_VEL
LIN {X 0,Y 234.917,Z 276.214,A -85,B 0,C 180,E1 -19654.641,E2 -19654.641} C_VEL
LIN {X 0,Y 234.908,Z 276.219,A -85,B 0,C 180,E1 -19658.937,E2 -19658.937} C_VEL
LIN {X 0,Y 234.859,Z 276.186,A -85,B 0,C 180,E1 -19664.098,E2 -19664.098} C_VEL
LIN {X 0,Y 234.852,Z 276.231,A -85,B 0,C 180,E1 -19668.827,E2 -19668.827} C_VEL
LIN {X 0,Y 234.916,Z 276.201,A -85,B 0,C 180,E1 -19671.08,E2 -19671.08} C_VEL
LIN {X 0,Y 234.921,Z 276.215,A -85,B 0,C 180,E1 -19675.362,E2 -19675.362} C_VEL
LIN {X 0,Y 234.893,Z 276.203,A -85,B 0,C 180,E1 -19679.428,E2 -19679.428} C_VEL
LIN {X 0,Y 234.94,Z 276.209,A -85,B 0,C 180,E1 -19683.823,E2 -19683.823} C_VEL
LIN {X 0,Y 234.958,Z 276.458,A -85,B 0,C 180,E1 -19686.536,E2 -19686.536} C_VEL
LIN {X 0,Y 235.216,Z 277.551,A -85,B 0,C 180,E1 -19686.822,E2 -19686.822} C_VEL
LIN {X 0,Y 242.327,Z 291.593,A -85,B 0,C 180,E1 -19688.216,E2 -19688.216} C_VEL
LIN {X 0,Y 249.795,Z 308.622,A -85,B 0,C 180,E1 -19689.635,E2 -19689.635} C_VEL
LIN {X 0,Y 248.461,Z 361.263,A -85,B 0,C 180,E1 -19691.16,E2 -19691.16} C_VEL
LIN {X 0,Y 247.875,Z 374.319,A -85,B 0,C 180,E1 -19691.797,E2 -19691.797} C_VEL
LIN {X 0,Y 247.165,Z 386.545,A -85,B 0,C 180,E1 -19692.737,E2 -19692.737} C_VEL
LIN {X 0,Y 245.856,Z 399.143,A -85,B 0,C 180,E1 -19694.031,E2 -19694.031} C_VEL
LIN {X 0,Y 244.429,Z 409.643,A -85,B 0,C 180,E1 -19695.43,E2 -19695.43} C_VEL
LIN {X 0,Y 242.834,Z 420.349,A -85,B 0,C 180,E1 -19697.252,E2 -19697.252} C_VEL
LIN {X 0,Y 241.084,Z 430.836,A -85,B 0,C 180,E1 -19699.503,E2 -19699.503} C_VEL
LIN {X 0,Y 239.536,Z 438.607,A -85,B 0,C 180,E1 -19701.565,E2 -19701.565} C_VEL
LIN {X 0,Y 237.976,Z 446.203,A -85,B 0,C 180,E1 -19704.068,E2 -19704.068} C_VEL
LIN {X 0,Y 236.824,Z 452.288,A -85,B 0,C 180,E1 -19706.598,E2 -19706.598} C_VEL
LIN {X 0,Y 235.882,Z 457.144,A -85,B 0,C 180,E1 -19709.147,E2 -19709.147} C_VEL
LIN {X 0,Y 235.138,Z 460.915,A -85,B 0,C 180,E1 -19711.713,E2 -19711.713} C_VEL
LIN {X 0,Y 234.853,Z 462.863,A -85,B 0,C 180,E1 -19713.432,E2 -19713.432} C_VEL
LIN {X 0,Y 234.846,Z 464.384,A -85,B 0,C 180,E1 -19715.151,E2 -19715.151} C_VEL
LIN {X 0,Y 234.796,Z 465.486,A -85,B 0,C 180,E1 -19716.877,E2 -19716.877} C_VEL
LIN {X 0,Y 234.993,Z 466.538,A -85,B 0,C 180,E1 -19720.338,E2 -19720.338} C_VEL
LIN {X 0,Y 235.298,Z 466.493,A -85,B 0,C 180,E1 -19722.069,E2 -19722.069} C_VEL
LIN {X 0,Y 235.739,Z 466.015,A -85,B 0,C 180,E1 -19723.799,E2 -19723.799} C_VEL
LIN {X 0,Y 236.265,Z 465.149,A -85,B 0,C 180,E1 -19725.529,E2 -19725.529} C_VEL
LIN {X 0,Y 237.037,Z 463.881,A -85,B 0,C 180,E1 -19727.247,E2 -19727.247} C_VEL
LIN {X 0,Y 238.374,Z 461.164,A -85,B 0,C 180,E1 -19729.819,E2 -19729.819} C_VEL
LIN {X 0,Y 240.031,Z 457.408,A -85,B 0,C 180,E1 -19732.373,E2 -19732.373} C_VEL
LIN {X 0,Y 242.03,Z 452.499,A -85,B 0,C 180,E1 -19734.901,E2 -19734.901} C_VEL
LIN {X 0,Y 244.411,Z 446.262,A -85,B 0,C 180,E1 -19737.392,E2 -19737.392} C_VEL
LIN {X 0,Y 247.092,Z 438.378,A -85,B 0,C 180,E1 -19739.851,E2 -19739.851} C_VEL
LIN {X 0,Y 249.605,Z 430.28,A -85,B 0,C 180,E1 -19741.866,E2 -19741.866} C_VEL
LIN {X 0,Y 252.237,Z 420.338,A -85,B 0,C 180,E1 -19743.866,E2 -19743.866} C_VEL
LIN {X 0,Y 254.494,Z 410.42,A -85,B 0,C 180,E1 -19745.445,E2 -19745.445} C_VEL
LIN {X 0,Y 256.23,Z 401.307,A -85,B 0,C 180,E1 -19746.624,E2 -19746.624} C_VEL
LIN {X 0,Y 258.122,Z 389.068,A -85,B 0,C 180,E1 -19747.851,E2 -19747.851} C_VEL
LIN {X 0,Y 259.344,Z 376.653,A -85,B 0,C 180,E1 -19748.792,E2 -19748.792} C_VEL
LIN {X 0,Y 260.112,Z 363.947,A -85,B 0,C 180,E1 -19749.443,E2 -19749.443} C_VEL
LIN {X 0,Y 261.356,Z 325.283,A -85,B 0,C 180,E1 -19750.572,E2 -19750.572} C_VEL
LIN {X 0,Y 261.393,Z 321.327,A -85,B 0,C 180,E1 -19750.7,E2 -19750.7} C_VEL
LIN {X 0,Y 254.669,Z 308.356,A -85,B 0,C 180,E1 -19752.302,E2 -19752.302} C_VEL
LIN {X 0,Y 247.037,Z 295.523,A -85,B 0,C 180,E1 -19754.207,E2 -19754.207} C_VEL
LIN {X 0,Y 242.055,Z 287.915,A -85,B 0,C 180,E1 -19755.52,E2 -19755.52} C_VEL
LIN {X 0,Y 239.985,Z 284.799,A -85,B 0,C 180,E1 -19756.088,E2 -19756.088} C_VEL
LIN {X 0,Y 237.762,Z 281.267,A -85,B 0,C 180,E1 -19756.722,E2 -19756.722} C_VEL
LIN {X 0,Y 235.596,Z 278.643,A -85,B 0,C 180,E1 -19757.324,E2 -19757.324} C_VEL
LIN {X 0,Y 234.937,Z 276.753,A -85,B 0,C 180,E1 -19757.692,E2 -19757.692} C_VEL
LIN {X 0,Y 234.898,Z 276.27,A -85,B 0,C 180,E1 -19758.068,E2 -19758.068} C_VEL
LIN {X 0,Y 234.918,Z 276.195,A -85,B 0,C 180,E1 -19761.078,E2 -19761.078} C_VEL
LIN {X 0,Y 234.922,Z 276.22,A -85,B 0,C 180,E1 -19765.36,E2 -19765.36} C_VEL
LIN {X 0,Y 234.894,Z 276.179,A -85,B 0,C 180,E1 -19769.426,E2 -19769.426} C_VEL
LIN {X 0,Y 234.967,Z 276.221,A -85,B 0,C 180,E1 -19773.806,E2 -19773.806} C_VEL
LIN {X 0,Y 234.992,Z 276.156,A -85,B 0,C 180,E1 -19778.967,E2 -19778.967} C_VEL
LIN {X 0,Y 235.095,Z 276.201,A -85,B 0,C 180,E1 -19783.059,E2 -19783.059} C_VEL
LIN {X 0,Y 235.111,Z 276.2,A -85,B 0,C 180,E1 -19787.921,E2 -19787.921} C_VEL
LIN {X 0,Y 235.308,Z 276.157,A -85,B 0,C 180,E1 -19791.411,E2 -19791.411} C_VEL
LIN {X 0,Y 235.343,Z 276.169,A -85,B 0,C 180,E1 -19793.139,E2 -19793.139} C_VEL
LIN {X 0,Y 235.573,Z 276.138,A -85,B 0,C 180,E1 -19798.29,E2 -19798.29} C_VEL
LIN {X 0,Y 235.574,Z 276.122,A -85,B 0,C 180,E1 -19801.709,E2 -19801.709} C_VEL
LIN {X 0,Y 235.343,Z 276.153,A -85,B 0,C 180,E1 -19806.86,E2 -19806.86} C_VEL
LIN {X 0,Y 235.207,Z 276.186,A -85,B 0,C 180,E1 -19810.328,E2 -19810.328} C_VEL
LIN {X 0,Y 235.083,Z 276.203,A -85,B 0,C 180,E1 -19815.608,E2 -19815.608} C_VEL
LIN {X 0,Y 234.99,Z 276.209,A -85,B 0,C 180,E1 -19819.207,E2 -19819.207} C_VEL
LIN {X 0,Y 234.942,Z 276.214,A -85,B 0,C 180,E1 -19822.884,E2 -19822.884} C_VEL
LIN {X 0,Y 234.915,Z 276.215,A -85,B 0,C 180,E1 -19823.709,E2 -19823.709} C_VEL
LIN {X 0,Y 234.244,Z 276.302,A -85,B 0,C 180,E1 -19825.139,E2 -19825.139} C_VEL
LIN {X 0,Y 231.374,Z 276.658,A -85,B 0,C 180,E1 -19827.471,E2 -19827.471} C_VEL
LIN {X 0,Y 228.944,Z 276.959,A -85,B 0,C 180,E1 -19829.372,E2 -19829.372} C_VEL
LIN {X 0,Y 227.919,Z 277.097,A -85,B 0,C 180,E1 -19830.849,E2 -19830.849} C_VEL
LIN {X 0,Y 227.844,Z 277.096,A -85,B 0,C 180,E1 -19831.349,E2 -19831.349} C_VEL
LIN {X 0,Y 227.878,Z 277.092,A -85,B 0,C 180,E1 -19835.872,E2 -19835.872} C_VEL
LIN {X 0,Y 227.888,Z 277.26,A -85,B 0,C 180,E1 -19839.254,E2 -19839.254} C_VEL
LIN {X 0,Y 230.977,Z 286.857,A -85,B 0,C 180,E1 -19843.805,E2 -19843.805} C_VEL
LIN {X 0,Y 234.037,Z 297.287,A -85,B 0,C 180,E1 -19848.171,E2 -19848.171} C_VEL
LIN {X 0,Y 235.342,Z 302.065,A -85,B 0,C 180,E1 -19849.927,E2 -19849.927} C_VEL
LIN {X 0,Y 241.066,Z 313.7,A -85,B 0,C 180,E1 -19851.668,E2 -19851.668} C_VEL
LIN {X 0,Y 246.081,Z 324.981,A -85,B 0,C 180,E1 -19853.099,E2 -19853.099} C_VEL
LIN {X 0,Y 246.947,Z 327.551,A -85,B 0,C 180,E1 -19853.36,E2 -19853.36} C_VEL
LIN {X 0,Y 250.724,Z 355.819,A -85,B 0,C 180,E1 -19855.076,E2 -19855.076} C_VEL
LIN {X 0,Y 253.035,Z 378.688,A -85,B 0,C 180,E1 -19856.272,E2 -19856.272} C_VEL
LIN {X 0,Y 253.243,Z 384.325,A -85,B 0,C 180,E1 -19856.501,E2 -19856.501} C_VEL
LIN {X 0,Y 251.69,Z 416.219,A -85,B 0,C 180,E1 -19857.409,E2 -19857.409} C_VEL
LIN {X 0,Y 250.295,Z 429.364,A -85,B 0,C 180,E1 -19858.055,E2 -19858.055} C_VEL
LIN {X 0,Y 248.233,Z 442.415,A -85,B 0,C 180,E1 -19859.007,E2 -19859.007} C_VEL
LIN {X 0,Y 245.611,Z 454.265,A -85,B 0,C 180,E1 -19860.187,E2 -19860.187} C_VEL
LIN {X 0,Y 242.535,Z 465.692,A -85,B 0,C 180,E1 -19861.673,E2 -19861.673} C_VEL
LIN {X 0,Y 239.41,Z 476.033,A -85,B 0,C 180,E1 -19863.406,E2 -19863.406} C_VEL
LIN {X 0,Y 236.428,Z 485.37,A -85,B 0,C 180,E1 -19865.407,E2 -19865.407} C_VEL
LIN {X 0,Y 233.275,Z 494.484,A -85,B 0,C 180,E1 -19867.877,E2 -19867.877} C_VEL
LIN {X 0,Y 230.785,Z 501.891,A -85,B 0,C 180,E1 -19870.428,E2 -19870.428} C_VEL
LIN {X 0,Y 229.345,Z 506.006,A -85,B 0,C 180,E1 -19872.155,E2 -19872.155} C_VEL
LIN {X 0,Y 227.866,Z 511.179,A -85,B 0,C 180,E1 -19874.801,E2 -19874.801} C_VEL
LIN {X 0,Y 226.771,Z 515.235,A -85,B 0,C 180,E1 -19877.47,E2 -19877.47} C_VEL
LIN {X 0,Y 226.269,Z 519.104,A -85,B 0,C 180,E1 -19881.065,E2 -19881.065} C_VEL
LIN {X 0,Y 226.436,Z 520.682,A -85,B 0,C 180,E1 -19883.314,E2 -19883.314} C_VEL
LIN {X 0,Y 226.857,Z 521.817,A -85,B 0,C 180,E1 -19886.447,E2 -19886.447} C_VEL
LIN {X 0,Y 227.122,Z 521.901,A -85,B 0,C 180,E1 -19888.226,E2 -19888.226} C_VEL
LIN {X 0,Y 227.256,Z 521.562,A -85,B 0,C 180,E1 -19889.999,E2 -19889.999} C_VEL
LIN {X 0,Y 227.188,Z 520.74,A -85,B 0,C 180,E1 -19891.772,E2 -19891.772} C_VEL
LIN {X 0,Y 226.997,Z 519.467,A -85,B 0,C 180,E1 -19893.549,E2 -19893.549} C_VEL
LIN {X 0,Y 226.72,Z 517.749,A -85,B 0,C 180,E1 -19895.335,E2 -19895.335} C_VEL
LIN {X 0,Y 226.469,Z 514.282,A -85,B 0,C 180,E1 -19898.027,E2 -19898.027} C_VEL
LIN {X 0,Y 226.567,Z 509.706,A -85,B 0,C 180,E1 -19900.725,E2 -19900.725} C_VEL
LIN {X 0,Y 227.141,Z 503.913,A -85,B 0,C 180,E1 -19903.417,E2 -19903.417} C_VEL
LIN {X 0,Y 228.136,Z 496.667,A -85,B 0,C 180,E1 -19906.095,E2 -19906.095} C_VEL
LIN {X 0,Y 229.516,Z 489.174,A -85,B 0,C 180,E1 -19908.333,E2 -19908.333} C_VEL
LIN {X 0,Y 231.136,Z 480.426,A -85,B 0,C 180,E1 -19910.466,E2 -19910.466} C_VEL
LIN {X 0,Y 232.995,Z 470.701,A -85,B 0,C 180,E1 -19912.383,E2 -19912.383} C_VEL
LIN {X 0,Y 235.098,Z 460.14,A -85,B 0,C 180,E1 -19914.034,E2 -19914.034} C_VEL
LIN {X 0,Y 236.946,Z 448.452,A -85,B 0,C 180,E1 -19915.471,E2 -19915.471} C_VEL
LIN {X 0,Y 238.536,Z 436.313,A -85,B 0,C 180,E1 -19916.58,E2 -19916.58} C_VEL
LIN {X 0,Y 239.825,Z 423.142,A -85,B 0,C 180,E1 -19917.427,E2 -19917.427} C_VEL
LIN {X 0,Y 240.423,Z 410.524,A -85,B 0,C 180,E1 -19917.942,E2 -19917.942} C_VEL
LIN {X 0,Y 241.265,Z 378.577,A -85,B 0,C 180,E1 -19918.871,E2 -19918.871} C_VEL
LIN {X 0,Y 238.118,Z 339.063,A -85,B 0,C 180,E1 -19920.508,E2 -19920.508} C_VEL
LIN {X 0,Y 234.481,Z 306.732,A -85,B 0,C 180,E1 -19922.052,E2 -19922.052} C_VEL
LIN {X 0,Y 234.234,Z 305.453,A -85,B 0,C 180,E1 -19922.197,E2 -19922.197} C_VEL
LIN {X 0,Y 232.356,Z 295.62,A -85,B 0,C 180,E1 -19925.248,E2 -19925.248} C_VEL
LIN {X 0,Y 229.925,Z 285.023,A -85,B 0,C 180,E1 -19928.79,E2 -19928.79} C_VEL
LIN {X 0,Y 227.835,Z 277.206,A -85,B 0,C 180,E1 -19931.646,E2 -19931.646} C_VEL
LIN {X 0,Y 227.805,Z 277.071,A -85,B 0,C 180,E1 -19935.198,E2 -19935.198} C_VEL
LIN {X 0,Y 227.794,Z 277.109,A -85,B 0,C 180,E1 -19939.617,E2 -19939.617} C_VEL
LIN {X 0,Y 227.874,Z 277.1,A -85,B 0,C 180,E1 -19944.127,E2 -19944.127} C_VEL
LIN {X 0,Y 227.846,Z 277.087,A -85,B 0,C 180,E1 -19948.374,E2 -19948.374} C_VEL
LIN {X 0,Y 227.844,Z 277.103,A -85,B 0,C 180,E1 -19952.44,E2 -19952.44} C_VEL
LIN {X 0,Y 227.882,Z 277.092,A -85,B 0,C 180,E1 -19956.364,E2 -19956.364} C_VEL
LIN {X 0,Y 227.884,Z 277.093,A -85,B 0,C 180,E1 -19960.17,E2 -19960.17} C_VEL
LIN {X 0,Y 228.009,Z 277.076,A -85,B 0,C 180,E1 -19963.895,E2 -19963.895} C_VEL
LIN {X 0,Y 228.047,Z 277.074,A -85,B 0,C 180,E1 -19967.542,E2 -19967.542} C_VEL
LIN {X 0,Y 228.243,Z 277.037,A -85,B 0,C 180,E1 -19971.144,E2 -19971.144} C_VEL
LIN {X 0,Y 228.29,Z 277.043,A -85,B 0,C 180,E1 -19972.927,E2 -19972.927} C_VEL
LIN {X 0,Y 228.526,Z 277.001,A -85,B 0,C 180,E1 -19978.238,E2 -19978.238} C_VEL
LIN {X 0,Y 228.523,Z 277.012,A -85,B 0,C 180,E1 -19981.763,E2 -19981.763} C_VEL
LIN {X 0,Y 228.283,Z 277.035,A -85,B 0,C 180,E1 -19987.074,E2 -19987.074} C_VEL
LIN {X 0,Y 228.119,Z 277.058,A -85,B 0,C 180,E1 -19990.653,E2 -19990.653} C_VEL
LIN {X 0,Y 228.023,Z 277.078,A -85,B 0,C 180,E1 -19994.275,E2 -19994.275} C_VEL
LIN {X 0,Y 227.922,Z 277.072,A -85,B 0,C 180,E1 -19997.96,E2 -19997.96} C_VEL
LIN {X 0,Y 227.885,Z 277.098,A -85,B 0,C 180,E1 -20002.306,E2 -20002.306} C_VEL
LIN {X 0,Y 227.863,Z 277.085,A -85,B 0,C 180,E1 -20006.567,E2 -20006.567} C_VEL
LIN {X 0,Y 227.864,Z 277.101,A -85,B 0,C 180,E1 -20010.28,E2 -20010.28} C_VEL
LIN {X 0,Y 227.871,Z 277.085,A -85,B 0,C 180,E1 -20013.722,E2 -20013.722} C_VEL
LIN {X 0,Y 227.836,Z 277.102,A -85,B 0,C 180,E1 -20018.093,E2 -20018.093} C_VEL
LIN {X 0,Y 227.78,Z 277.061,A -85,B 0,C 180,E1 -20022.75,E2 -20022.75} C_VEL
LIN {X 0,Y 227.807,Z 277.077,A -85,B 0,C 180,E1 -20025.201,E2 -20025.201} C_VEL
LIN {X 0,Y 227.798,Z 277.104,A -85,B 0,C 180,E1 -20029.619,E2 -20029.619} C_VEL
LIN {X 0,Y 227.863,Z 277.073,A -85,B 0,C 180,E1 -20034.127,E2 -20034.127} C_VEL
LIN {X 0,Y 227.853,Z 277.087,A -85,B 0,C 180,E1 -20038.377,E2 -20038.377} C_VEL
LIN {X 0,Y 227.84,Z 277.106,A -85,B 0,C 180,E1 -20042.441,E2 -20042.441} C_VEL
LIN {X 0,Y 227.903,Z 277.316,A -85,B 0,C 180,E1 -20045.581,E2 -20045.581} C_VEL
LIN {X 0,Y 228.164,Z 278.41,A -85,B 0,C 180,E1 -20045.882,E2 -20045.882} C_VEL
LIN {X 0,Y 236.506,Z 294.724,A -85,B 0,C 180,E1 -20047.593,E2 -20047.593} C_VEL
LIN {X 0,Y 243.406,Z 310.572,A -85,B 0,C 180,E1 -20048.964,E2 -20048.964} C_VEL
LIN {X 0,Y 242.002,Z 360.88,A -85,B 0,C 180,E1 -20050.446,E2 -20050.446} C_VEL
LIN {X 0,Y 241.47,Z 374.052,A -85,B 0,C 180,E1 -20051.079,E2 -20051.079} C_VEL
LIN {X 0,Y 240.723,Z 386.611,A -85,B 0,C 180,E1 -20052.04,E2 -20052.04} C_VEL
LIN {X 0,Y 239.35,Z 399.379,A -85,B 0,C 180,E1 -20053.365,E2 -20053.365} C_VEL
LIN {X 0,Y 237.856,Z 410.002,A -85,B 0,C 180,E1 -20054.799,E2 -20054.799} C_VEL
LIN {X 0,Y 236.185,Z 420.825,A -85,B 0,C 180,E1 -20056.668,E2 -20056.668} C_VEL
LIN {X 0,Y 234.505,Z 430.5,A -85,B 0,C 180,E1 -20058.768,E2 -20058.768} C_VEL
LIN {X 0,Y 232.894,Z 438.463,A -85,B 0,C 180,E1 -20060.885,E2 -20060.885} C_VEL
LIN {X 0,Y 231.256,Z 446.286,A -85,B 0,C 180,E1 -20063.457,E2 -20063.457} C_VEL
LIN {X 0,Y 230.191,Z 451.571,A -85,B 0,C 180,E1 -20065.623,E2 -20065.623} C_VEL
LIN {X 0,Y 229.164,Z 456.761,A -85,B 0,C 180,E1 -20068.243,E2 -20068.243} C_VEL
LIN {X 0,Y 228.342,Z 460.823,A -85,B 0,C 180,E1 -20070.882,E2 -20070.882} C_VEL
LIN {X 0,Y 227.798,Z 463.857,A -85,B 0,C 180,E1 -20073.538,E2 -20073.538} C_VEL
LIN {X 0,Y 227.807,Z 465.337,A -85,B 0,C 180,E1 -20075.311,E2 -20075.311} C_VEL
LIN {X 0,Y 227.804,Z 467.093,A -85,B 0,C 180,E1 -20078.874,E2 -20078.874} C_VEL
LIN {X 0,Y 227.984,Z 467.407,A -85,B 0,C 180,E1 -20080.659,E2 -20080.659} C_VEL
LIN {X 0,Y 228.342,Z 467.318,A -85,B 0,C 180,E1 -20082.442,E2 -20082.442} C_VEL
LIN {X 0,Y 229.39,Z 465.915,A -85,B 0,C 180,E1 -20086.007,E2 -20086.007} C_VEL
LIN {X 0,Y 230.24,Z 464.618,A -85,B 0,C 180,E1 -20087.773,E2 -20087.773} C_VEL
LIN {X 0,Y 231.661,Z 461.848,A -85,B 0,C 180,E1 -20090.419,E2 -20090.419} C_VEL
LIN {X 0,Y 233.418,Z 458.036,A -85,B 0,C 180,E1 -20093.043,E2 -20093.043} C_VEL
LIN {X 0,Y 235.566,Z 453.06,A -85,B 0,C 180,E1 -20095.633,E2 -20095.633} C_VEL
LIN {X 0,Y 238.063,Z 446.723,A -85,B 0,C 180,E1 -20098.187,E2 -20098.187} C_VEL
LIN {X 0,Y 240.906,Z 438.75,A -85,B 0,C 180,E1 -20100.699,E2 -20100.699} C_VEL
LIN {X 0,Y 243.536,Z 430.556,A -85,B 0,C 180,E1 -20102.758,E2 -20102.758} C_VEL
LIN {X 0,Y 246.301,Z 420.456,A -85,B 0,C 180,E1 -20104.798,E2 -20104.798} C_VEL
LIN {X 0,Y 248.925,Z 408.904,A -85,B 0,C 180,E1 -20106.615,E2 -20106.615} C_VEL
LIN {X 0,Y 251.136,Z 397.451,A -85,B 0,C 180,E1 -20108,E2 -20108} C_VEL
LIN {X 0,Y 252.711,Z 386.902,A -85,B 0,C 180,E1 -20108.982,E2 -20108.982} C_VEL
LIN {X 0,Y 253.754,Z 374.037,A -85,B 0,C 180,E1 -20109.905,E2 -20109.905} C_VEL
LIN {X 0,Y 254.421,Z 361.001,A -85,B 0,C 180,E1 -20110.495,E2 -20110.495} C_VEL
LIN {X 0,Y 255.664,Z 323.748,A -85,B 0,C 180,E1 -20111.586,E2 -20111.586} C_VEL
LIN {X 0,Y 249.519,Z 311.899,A -85,B 0,C 180,E1 -20113.121,E2 -20113.121} C_VEL
LIN {X 0,Y 242.494,Z 299.964,A -85,B 0,C 180,E1 -20114.959,E2 -20114.959} C_VEL
LIN {X 0,Y 235.849,Z 289.776,A -85,B 0,C 180,E1 -20116.808,E2 -20116.808} C_VEL
LIN {X 0,Y 232.903,Z 285.548,A -85,B 0,C 180,E1 -20117.668,E2 -20117.668} C_VEL
LIN {X 0,Y 230.347,Z 281.701,A -85,B 0,C 180,E1 -20118.45,E2 -20118.45} C_VEL
LIN {X 0,Y 228.403,Z 279.202,A -85,B 0,C 180,E1 -20119.049,E2 -20119.049} C_VEL
LIN {X 0,Y 227.868,Z 277.573,A -85,B 0,C 180,E1 -20119.417,E2 -20119.417} C_VEL
LIN {X 0,Y 227.822,Z 277.107,A -85,B 0,C 180,E1 -20120.117,E2 -20120.117} C_VEL
LIN {X 0,Y 227.864,Z 277.075,A -85,B 0,C 180,E1 -20124.125,E2 -20124.125} C_VEL
LIN {X 0,Y 227.853,Z 277.062,A -85,B 0,C 180,E1 -20128.374,E2 -20128.374} C_VEL
LIN {X 0,Y 227.851,Z 277.089,A -85,B 0,C 180,E1 -20132.44,E2 -20132.44} C_VEL
LIN {X 0,Y 227.893,Z 277.051,A -85,B 0,C 180,E1 -20136.365,E2 -20136.365} C_VEL
LIN {X 0,Y 227.932,Z 277.048,A -85,B 0,C 180,E1 -20140.173,E2 -20140.173} C_VEL
LIN {X 0,Y 228.055,Z 277.071,A -85,B 0,C 180,E1 -20143.897,E2 -20143.897} C_VEL
LIN {X 0,Y 228.069,Z 277.074,A -85,B 0,C 180,E1 -20147.543,E2 -20147.543} C_VEL
LIN {X 0,Y 228.25,Z 277.034,A -85,B 0,C 180,E1 -20151.143,E2 -20151.143} C_VEL
LIN {X 0,Y 228.296,Z 277.046,A -85,B 0,C 180,E1 -20152.926,E2 -20152.926} C_VEL
LIN {X 0,Y 228.531,Z 277.014,A -85,B 0,C 180,E1 -20158.237,E2 -20158.237} C_VEL
LIN {X 0,Y 228.532,Z 276.999,A -85,B 0,C 180,E1 -20161.762,E2 -20161.762} C_VEL
LIN {X 0,Y 228.295,Z 277.029,A -85,B 0,C 180,E1 -20167.073,E2 -20167.073} C_VEL
LIN {X 0,Y 228.138,Z 277.067,A -85,B 0,C 180,E1 -20170.651,E2 -20170.651} C_VEL
LIN {X 0,Y 228.036,Z 277.067,A -85,B 0,C 180,E1 -20174.274,E2 -20174.274} C_VEL
LIN {X 0,Y 227.968,Z 277.078,A -85,B 0,C 180,E1 -20177.956,E2 -20177.956} C_VEL
LIN {X 0,Y 227.917,Z 277.086,A -85,B 0,C 180,E1 -20182.322,E2 -20182.322} C_VEL
LIN {X 0,Y 227.918,Z 277.064,A -85,B 0,C 180,E1 -20186.591,E2 -20186.591} C_VEL
LIN {X 0,Y 227.844,Z 277.096,A -85,B 0,C 180,E1 -20191.349,E2 -20191.349} C_VEL
LIN {X 0,Y 227.172,Z 277.178,A -85,B 0,C 180,E1 -20192.33,E2 -20192.33} C_VEL
LIN {X 0,Y 224.31,Z 277.528,A -85,B 0,C 180,E1 -20193.868,E2 -20193.868} C_VEL
LIN {X 0,Y 221.432,Z 277.887,A -85,B 0,C 180,E1 -20195.444,E2 -20195.444} C_VEL
LIN {X 0,Y 220.778,Z 277.974,A -85,B 0,C 180,E1 -20196.468,E2 -20196.468} C_VEL
LIN {X 0,Y 220.847,Z 278.185,A -85,B 0,C 180,E1 -20197.697,E2 -20197.697} C_VEL
LIN {X 0,Y 223.932,Z 287.573,A -85,B 0,C 180,E1 -20202.436,E2 -20202.436} C_VEL
LIN {X 0,Y 226.59,Z 296.573,A -85,B 0,C 180,E1 -20206.446,E2 -20206.446} C_VEL
LIN {X 0,Y 227.883,Z 300.913,A -85,B 0,C 180,E1 -20208.12,E2 -20208.12} C_VEL
LIN {X 0,Y 234.214,Z 313.226,A -85,B 0,C 180,E1 -20210.173,E2 -20210.173} C_VEL
LIN {X 0,Y 240.403,Z 326.734,A -85,B 0,C 180,E1 -20212.037,E2 -20212.037} C_VEL
LIN {X 0,Y 241.642,Z 330.121,A -85,B 0,C 180,E1 -20212.419,E2 -20212.419} C_VEL
LIN {X 0,Y 245.211,Z 357.863,A -85,B 0,C 180,E1 -20214.152,E2 -20214.152} C_VEL
LIN {X 0,Y 247.402,Z 380.71,A -85,B 0,C 180,E1 -20215.379,E2 -20215.379} C_VEL
LIN {X 0,Y 247.4,Z 387.605,A -85,B 0,C 180,E1 -20215.626,E2 -20215.626} C_VEL
LIN {X 0,Y 245.922,Z 415.939,A -85,B 0,C 180,E1 -20216.457,E2 -20216.457} C_VEL
LIN {X 0,Y 244.431,Z 429.22,A -85,B 0,C 180,E1 -20217.132,E2 -20217.132} C_VEL
LIN {X 0,Y 242.391,Z 441.523,A -85,B 0,C 180,E1 -20218.052,E2 -20218.052} C_VEL
LIN {X 0,Y 239.493,Z 454.171,A -85,B 0,C 180,E1 -20219.344,E2 -20219.344} C_VEL
LIN {X 0,Y 236.326,Z 465.458,A -85,B 0,C 180,E1 -20220.858,E2 -20220.858} C_VEL
LIN {X 0,Y 233.094,Z 475.665,A -85,B 0,C 180,E1 -20222.626,E2 -20222.626} C_VEL
LIN {X 0,Y 229.975,Z 484.903,A -85,B 0,C 180,E1 -20224.669,E2 -20224.669} C_VEL
LIN {X 0,Y 226.676,Z 493.949,A -85,B 0,C 180,E1 -20227.197,E2 -20227.197} C_VEL
LIN {X 0,Y 224.062,Z 501.297,A -85,B 0,C 180,E1 -20229.816,E2 -20229.816} C_VEL
LIN {X 0,Y 222.007,Z 507.23,A -85,B 0,C 180,E1 -20232.498,E2 -20232.498} C_VEL
LIN {X 0,Y 220.528,Z 511.967,A -85,B 0,C 180,E1 -20235.229,E2 -20235.229} C_VEL
LIN {X 0,Y 219.559,Z 515.634,A -85,B 0,C 180,E1 -20237.991,E2 -20237.991} C_VEL
LIN {X 0,Y 219.217,Z 518.329,A -85,B 0,C 180,E1 -20240.775,E2 -20240.775} C_VEL
LIN {X 0,Y 219.362,Z 519.978,A -85,B 0,C 180,E1 -20243.309,E2 -20243.309} C_VEL
LIN {X 0,Y 219.782,Z 520.972,A -85,B 0,C 180,E1 -20246.333,E2 -20246.333} C_VEL
LIN {X 0,Y 220.068,Z 521.042,A -85,B 0,C 180,E1 -20248.169,E2 -20248.169} C_VEL
LIN {X 0,Y 220.206,Z 520.677,A -85,B 0,C 180,E1 -20249.999,E2 -20249.999} C_VEL
LIN {X 0,Y 220.136,Z 519.825,A -85,B 0,C 180,E1 -20251.829,E2 -20251.829} C_VEL
LIN {X 0,Y 219.92,Z 518.528,A -85,B 0,C 180,E1 -20253.664,E2 -20253.664} C_VEL
LIN {X 0,Y 219.51,Z 515.029,A -85,B 0,C 180,E1 -20257.012,E2 -20257.012} C_VEL
LIN {X 0,Y 219.442,Z 510.33,A -85,B 0,C 180,E1 -20260.144,E2 -20260.144} C_VEL
LIN {X 0,Y 220.034,Z 503.852,A -85,B 0,C 180,E1 -20263.388,E2 -20263.388} C_VEL
LIN {X 0,Y 221.012,Z 496.81,A -85,B 0,C 180,E1 -20266.154,E2 -20266.154} C_VEL
LIN {X 0,Y 222.551,Z 488.814,A -85,B 0,C 180,E1 -20268.67,E2 -20268.67} C_VEL
LIN {X 0,Y 224.483,Z 479.103,A -85,B 0,C 180,E1 -20271.101,E2 -20271.101} C_VEL
LIN {X 0,Y 226.449,Z 469.284,A -85,B 0,C 180,E1 -20273.067,E2 -20273.067} C_VEL
LIN {X 0,Y 228.545,Z 458.579,A -85,B 0,C 180,E1 -20274.769,E2 -20274.769} C_VEL
LIN {X 0,Y 230.511,Z 446.625,A -85,B 0,C 180,E1 -20276.236,E2 -20276.236} C_VEL
LIN {X 0,Y 232.115,Z 434.166,A -85,B 0,C 180,E1 -20277.376,E2 -20277.376} C_VEL
LIN {X 0,Y 233.406,Z 421.407,A -85,B 0,C 180,E1 -20278.186,E2 -20278.186} C_VEL
LIN {X 0,Y 234.035,Z 406.74,A -85,B 0,C 180,E1 -20278.753,E2 -20278.753} C_VEL
LIN {X 0,Y 234.858,Z 379.734,A -85,B 0,C 180,E1 -20279.552,E2 -20279.552} C_VEL
LIN {X 0,Y 231.879,Z 340.927,A -85,B 0,C 180,E1 -20281.209,E2 -20281.209} C_VEL
LIN {X 0,Y 228.288,Z 308.491,A -85,B 0,C 180,E1 -20282.797,E2 -20282.797} C_VEL
LIN {X 0,Y 226.924,Z 304.47,A -85,B 0,C 180,E1 -20283.209,E2 -20283.209} C_VEL
LIN {X 0,Y 224.684,Z 293.496,A -85,B 0,C 180,E1 -20286.803,E2 -20286.803} C_VEL
LIN {X 0,Y 222.463,Z 284.323,A -85,B 0,C 180,E1 -20290.039,E2 -20290.039} C_VEL
LIN {X 0,Y 220.761,Z 278.063,A -85,B 0,C 180,E1 -20292.464,E2 -20292.464} C_VEL
LIN {X 0,Y 220.738,Z 277.967,A -85,B 0,C 180,E1 -20297.076,E2 -20297.076} C_VEL
LIN {X 0,Y 220.775,Z 277.976,A -85,B 0,C 180,E1 -20300.457,E2 -20300.457} C_VEL
LIN {X 0,Y 220.819,Z 277.971,A -85,B 0,C 180,E1 -20302.792,E2 -20302.792} C_VEL
LIN {X 0,Y 220.804,Z 277.961,A -85,B 0,C 180,E1 -20307.242,E2 -20307.242} C_VEL
LIN {X 0,Y 220.793,Z 277.982,A -85,B 0,C 180,E1 -20311.481,E2 -20311.481} C_VEL
LIN {X 0,Y 220.837,Z 277.964,A -85,B 0,C 180,E1 -20315.562,E2 -20315.562} C_VEL
LIN {X 0,Y 220.842,Z 277.972,A -85,B 0,C 180,E1 -20319.509,E2 -20319.509} C_VEL
LIN {X 0,Y 220.968,Z 277.947,A -85,B 0,C 180,E1 -20323.367,E2 -20323.367} C_VEL
LIN {X 0,Y 221.054,Z 277.934,A -85,B 0,C 180,E1 -20329.003,E2 -20329.003} C_VEL
LIN {X 0,Y 221.228,Z 277.92,A -85,B 0,C 180,E1 -20332.7,E2 -20332.7} C_VEL
LIN {X 0,Y 221.459,Z 277.88,A -85,B 0,C 180,E1 -20338.182,E2 -20338.182} C_VEL
LIN {X 0,Y 221.456,Z 277.892,A -85,B 0,C 180,E1 -20341.819,E2 -20341.819} C_VEL
LIN {X 0,Y 221.221,Z 277.912,A -85,B 0,C 180,E1 -20347.301,E2 -20347.301} C_VEL
LIN {X 0,Y 221.045,Z 277.943,A -85,B 0,C 180,E1 -20350.998,E2 -20350.998} C_VEL
LIN {X 0,Y 220.953,Z 277.955,A -85,B 0,C 180,E1 -20354.742,E2 -20354.742} C_VEL
LIN {X 0,Y 220.862,Z 277.954,A -85,B 0,C 180,E1 -20358.555,E2 -20358.555} C_VEL
LIN {X 0,Y 220.831,Z 277.975,A -85,B 0,C 180,E1 -20362.646,E2 -20362.646} C_VEL
LIN {X 0,Y 220.82,Z 277.964,A -85,B 0,C 180,E1 -20366.986,E2 -20366.986} C_VEL
LIN {X 0,Y 220.813,Z 277.978,A -85,B 0,C 180,E1 -20370.76,E2 -20370.76} C_VEL
LIN {X 0,Y 220.788,Z 277.975,A -85,B 0,C 180,E1 -20374.958,E2 -20374.958} C_VEL
LIN {X 0,Y 220.797,Z 277.982,A -85,B 0,C 180,E1 -20377.277,E2 -20377.277} C_VEL
LIN {X 0,Y 220.741,Z 277.94,A -85,B 0,C 180,E1 -20381.96,E2 -20381.96} C_VEL
LIN {X 0,Y 220.75,Z 277.96,A -85,B 0,C 180,E1 -20385.542,E2 -20385.542} C_VEL
LIN {X 0,Y 220.779,Z 277.968,A -85,B 0,C 180,E1 -20390.459,E2 -20390.459} C_VEL
LIN {X 0,Y 220.823,Z 277.94,A -85,B 0,C 180,E1 -20392.795,E2 -20392.795} C_VEL
LIN {X 0,Y 220.81,Z 277.978,A -85,B 0,C 180,E1 -20397.245,E2 -20397.245} C_VEL
LIN {X 0,Y 220.795,Z 277.967,A -85,B 0,C 180,E1 -20401.482,E2 -20401.482} C_VEL
LIN {X 0,Y 220.859,Z 278.187,A -85,B 0,C 180,E1 -20404.559,E2 -20404.559} C_VEL
LIN {X 0,Y 221.067,Z 279.161,A -85,B 0,C 180,E1 -20404.856,E2 -20404.856} C_VEL
LIN {X 0,Y 230.062,Z 296.532,A -85,B 0,C 180,E1 -20406.805,E2 -20406.805} C_VEL
LIN {X 0,Y 236.876,Z 312.011,A -85,B 0,C 180,E1 -20408.221,E2 -20408.221} C_VEL
LIN {X 0,Y 235.579,Z 363.177,A -85,B 0,C 180,E1 -20409.799,E2 -20409.799} C_VEL
LIN {X 0,Y 234.949,Z 376.099,A -85,B 0,C 180,E1 -20410.469,E2 -20410.469} C_VEL
LIN {X 0,Y 234.182,Z 387.798,A -85,B 0,C 180,E1 -20411.407,E2 -20411.407} C_VEL
LIN {X 0,Y 232.873,Z 399.617,A -85,B 0,C 180,E1 -20412.662,E2 -20412.662} C_VEL
LIN {X 0,Y 231.319,Z 410.355,A -85,B 0,C 180,E1 -20414.132,E2 -20414.132} C_VEL
LIN {X 0,Y 229.562,Z 421.302,A -85,B 0,C 180,E1 -20416.05,E2 -20416.05} C_VEL
LIN {X 0,Y 227.624,Z 431.916,A -85,B 0,C 180,E1 -20418.424,E2 -20418.424} C_VEL
LIN {X 0,Y 225.941,Z 439.788,A -85,B 0,C 180,E1 -20420.602,E2 -20420.602} C_VEL
LIN {X 0,Y 224.261,Z 447.505,A -85,B 0,C 180,E1 -20423.252,E2 -20423.252} C_VEL
LIN {X 0,Y 222.735,Z 454.568,A -85,B 0,C 180,E1 -20426.383,E2 -20426.383} C_VEL
LIN {X 0,Y 221.771,Z 459.299,A -85,B 0,C 180,E1 -20429.093,E2 -20429.093} C_VEL
LIN {X 0,Y 220.993,Z 462.96,A -85,B 0,C 180,E1 -20431.823,E2 -20431.823} C_VEL
LIN {X 0,Y 220.745,Z 464.85,A -85,B 0,C 180,E1 -20433.651,E2 -20433.651} C_VEL
LIN {X 0,Y 220.75,Z 466.28,A -85,B 0,C 180,E1 -20435.481,E2 -20435.481} C_VEL
LIN {X 0,Y 220.794,Z 467.985,A -85,B 0,C 180,E1 -20439.158,E2 -20439.158} C_VEL
LIN {X 0,Y 221.008,Z 468.273,A -85,B 0,C 180,E1 -20441,E2 -20441} C_VEL
LIN {X 0,Y 221.376,Z 468.136,A -85,B 0,C 180,E1 -20442.84,E2 -20442.84} C_VEL
LIN {X 0,Y 222.534,Z 466.682,A -85,B 0,C 180,E1 -20446.514,E2 -20446.514} C_VEL
LIN {X 0,Y 223.443,Z 465.354,A -85,B 0,C 180,E1 -20448.333,E2 -20448.333} C_VEL
LIN {X 0,Y 224.97,Z 462.532,A -85,B 0,C 180,E1 -20451.055,E2 -20451.055} C_VEL
LIN {X 0,Y 226.836,Z 458.661,A -85,B 0,C 180,E1 -20453.752,E2 -20453.752} C_VEL
LIN {X 0,Y 229.144,Z 453.606,A -85,B 0,C 180,E1 -20456.406,E2 -20456.406} C_VEL
LIN {X 0,Y 231.766,Z 447.18,A -85,B 0,C 180,E1 -20459.024,E2 -20459.024} C_VEL
LIN {X 0,Y 234.787,Z 439.123,A -85,B 0,C 180,E1 -20461.59,E2 -20461.59} C_VEL
LIN {X 0,Y 237.516,Z 430.846,A -85,B 0,C 180,E1 -20463.693,E2 -20463.693} C_VEL
LIN {X 0,Y 240.145,Z 421.714,A -85,B 0,C 180,E1 -20465.567,E2 -20465.567} C_VEL
LIN {X 0,Y 242.589,Z 411.698,A -85,B 0,C 180,E1 -20467.212,E2 -20467.212} C_VEL
LIN {X 0,Y 244.839,Z 400.717,A -85,B 0,C 180,E1 -20468.632,E2 -20468.632} C_VEL
LIN {X 0,Y 246.719,Z 389.199,A -85,B 0,C 180,E1 -20469.778,E2 -20469.778} C_VEL
LIN {X 0,Y 247.882,Z 377.277,A -85,B 0,C 180,E1 -20470.7,E2 -20470.7} C_VEL
LIN {X 0,Y 248.694,Z 365.271,A -85,B 0,C 180,E1 -20471.31,E2 -20471.31} C_VEL
LIN {X 0,Y 250.018,Z 326.118,A -85,B 0,C 180,E1 -20472.511,E2 -20472.511} C_VEL
LIN {X 0,Y 242.988,Z 312.857,A -85,B 0,C 180,E1 -20474.361,E2 -20474.361} C_VEL
LIN {X 0,Y 234.715,Z 299.141,A -85,B 0,C 180,E1 -20476.681,E2 -20476.681} C_VEL
LIN {X 0,Y 228.633,Z 290.26,A -85,B 0,C 180,E1 -20478.504,E2 -20478.504} C_VEL
LIN {X 0,Y 226.318,Z 286.843,A -85,B 0,C 180,E1 -20479.243,E2 -20479.243} C_VEL
LIN {X 0,Y 224.098,Z 283.487,A -85,B 0,C 180,E1 -20479.979,E2 -20479.979} C_VEL
LIN {X 0,Y 221.513,Z 280.344,A -85,B 0,C 180,E1 -20480.833,E2 -20480.833} C_VEL
LIN {X 0,Y 220.894,Z 278.582,A -85,B 0,C 180,E1 -20481.216,E2 -20481.216} C_VEL
LIN {X 0,Y 220.821,Z 278.045,A -85,B 0,C 180,E1 -20481.639,E2 -20481.639} C_VEL
LIN {X 0,Y 220.805,Z 277.985,A -85,B 0,C 180,E1 -20485.848,E2 -20485.848} C_VEL
LIN {X 0,Y 220.834,Z 277.929,A -85,B 0,C 180,E1 -20489.389,E2 -20489.389} C_VEL
LIN {X 0,Y 220.874,Z 277.975,A -85,B 0,C 180,E1 -20493.546,E2 -20493.546} C_VEL
LIN {X 0,Y 220.865,Z 277.912,A -85,B 0,C 180,E1 -20497.551,E2 -20497.551} C_VEL
LIN {X 0,Y 220.983,Z 277.959,A -85,B 0,C 180,E1 -20502.572,E2 -20502.572} C_VEL
LIN {X 0,Y 221.008,Z 277.95,A -85,B 0,C 180,E1 -20507.138,E2 -20507.138} C_VEL
LIN {X 0,Y 221.191,Z 277.913,A -85,B 0,C 180,E1 -20510.858,E2 -20510.858} C_VEL
LIN {X 0,Y 221.235,Z 277.923,A -85,B 0,C 180,E1 -20512.699,E2 -20512.699} C_VEL
LIN {X 0,Y 221.464,Z 277.894,A -85,B 0,C 180,E1 -20518.181,E2 -20518.181} C_VEL
LIN {X 0,Y 221.466,Z 277.878,A -85,B 0,C 180,E1 -20521.818,E2 -20521.818} C_VEL
LIN {X 0,Y 221.232,Z 277.908,A -85,B 0,C 180,E1 -20527.3,E2 -20527.3} C_VEL
LIN {X 0,Y 221.059,Z 277.946,A -85,B 0,C 180,E1 -20530.996,E2 -20530.996} C_VEL
LIN {X 0,Y 220.989,Z 277.954,A -85,B 0,C 180,E1 -20536.632,E2 -20536.632} C_VEL
LIN {X 0,Y 220.877,Z 277.972,A -85,B 0,C 180,E1 -20540.487,E2 -20540.487} C_VEL
LIN {X 0,Y 220.844,Z 277.976,A -85,B 0,C 180,E1 -20544.437,E2 -20544.437} C_VEL
LIN {X 0,Y 220.797,Z 277.95,A -85,B 0,C 180,E1 -20548.519,E2 -20548.519} C_VEL
LIN {X 0,Y 220.809,Z 277.957,A -85,B 0,C 180,E1 -20552.757,E2 -20552.757} C_VEL
LIN {X 0,Y 220.778,Z 277.974,A -85,B 0,C 180,E1 -20556.468,E2 -20556.468} C_VEL
LIN {X 0,Y 220.645,Z 278.645,A -85,B 0,C 180,E1 -20557.475,E2 -20557.475} C_VEL
LIN {X 0,Y 220.145,Z 280.809,A -85,B 0,C 180,E1 -20558.642,E2 -20558.642} C_VEL
LIN {X 0,Y 218.33,Z 289.594,A -85,B 0,C 180,E1 -20561.839,E2 -20561.839} C_VEL
LIN {X 0,Y 218.604,Z 293.786,A -85,B 0,C 180,E1 -20563.608,E2 -20563.608} C_VEL
LIN {X 0,Y 220.253,Z 299.455,A -85,B 0,C 180,E1 -20566.048,E2 -20566.048} C_VEL
LIN {X 0,Y 224.923,Z 308.22,A -85,B 0,C 180,E1 -20567.741,E2 -20567.741} C_VEL
LIN {X 0,Y 227.423,Z 312.989,A -85,B 0,C 180,E1 -20568.573,E2 -20568.573} C_VEL
LIN {X 0,Y 231.853,Z 322.085,A -85,B 0,C 180,E1 -20570.004,E2 -20570.004} C_VEL
LIN {X 0,Y 236.363,Z 332.552,A -85,B 0,C 180,E1 -20571.423,E2 -20571.423} C_VEL
LIN {X 0,Y 239.685,Z 359.004,A -85,B 0,C 180,E1 -20573.136,E2 -20573.136} C_VEL
LIN {X 0,Y 241.797,Z 381.815,A -85,B 0,C 180,E1 -20574.402,E2 -20574.402} C_VEL
LIN {X 0,Y 241.716,Z 388.831,A -85,B 0,C 180,E1 -20574.647,E2 -20574.647} C_VEL
LIN {X 0,Y 240.359,Z 414.172,A -85,B 0,C 180,E1 -20575.397,E2 -20575.397} C_VEL
LIN {X 0,Y 238.842,Z 427.573,A -85,B 0,C 180,E1 -20576.071,E2 -20576.071} C_VEL
LIN {X 0,Y 236.57,Z 440.641,A -85,B 0,C 180,E1 -20577.042,E2 -20577.042} C_VEL
LIN {X 0,Y 233.888,Z 452.497,A -85,B 0,C 180,E1 -20578.274,E2 -20578.274} C_VEL
LIN {X 0,Y 230.549,Z 463.928,A -85,B 0,C 180,E1 -20579.802,E2 -20579.802} C_VEL
LIN {X 0,Y 227.149,Z 474.272,A -85,B 0,C 180,E1 -20581.595,E2 -20581.595} C_VEL
LIN {X 0,Y 224.184,Z 482.773,A -85,B 0,C 180,E1 -20583.466,E2 -20583.466} C_VEL
LIN {X 0,Y 220.636,Z 492.037,A -85,B 0,C 180,E1 -20586.038,E2 -20586.038} C_VEL
LIN {X 0,Y 217.773,Z 499.56,A -85,B 0,C 180,E1 -20588.711,E2 -20588.711} C_VEL
LIN {X 0,Y 215.154,Z 506.562,A -85,B 0,C 180,E1 -20591.921,E2 -20591.921} C_VEL
LIN {X 0,Y 213.625,Z 511.259,A -85,B 0,C 180,E1 -20594.74,E2 -20594.74} C_VEL
LIN {X 0,Y 212.579,Z 514.891,A -85,B 0,C 180,E1 -20597.59,E2 -20597.59} C_VEL
LIN {X 0,Y 212.158,Z 517.554,A -85,B 0,C 180,E1 -20600.465,E2 -20600.465} C_VEL
LIN {X 0,Y 212.299,Z 519.263,A -85,B 0,C 180,E1 -20603.278,E2 -20603.278} C_VEL
LIN {X 0,Y 212.708,Z 520.127,A -85,B 0,C 180,E1 -20606.21,E2 -20606.21} C_VEL
LIN {X 0,Y 213.013,Z 520.182,A -85,B 0,C 180,E1 -20608.109,E2 -20608.109} C_VEL
LIN {X 0,Y 213.158,Z 519.784,A -85,B 0,C 180,E1 -20609.999,E2 -20609.999} C_VEL
LIN {X 0,Y 213.083,Z 518.908,A -85,B 0,C 180,E1 -20611.889,E2 -20611.889} C_VEL
LIN {X 0,Y 212.844,Z 517.588,A -85,B 0,C 180,E1 -20613.786,E2 -20613.786} C_VEL
LIN {X 0,Y 212.446,Z 514.272,A -85,B 0,C 180,E1 -20617.051,E2 -20617.051} C_VEL
LIN {X 0,Y 212.389,Z 509.272,A -85,B 0,C 180,E1 -20620.485,E2 -20620.485} C_VEL
LIN {X 0,Y 213.067,Z 502.745,A -85,B 0,C 180,E1 -20623.835,E2 -20623.835} C_VEL
LIN {X 0,Y 214.131,Z 495.648,A -85,B 0,C 180,E1 -20626.688,E2 -20626.688} C_VEL
LIN {X 0,Y 215.587,Z 488.444,A -85,B 0,C 180,E1 -20629.024,E2 -20629.024} C_VEL
LIN {X 0,Y 217.38,Z 479.749,A -85,B 0,C 180,E1 -20631.327,E2 -20631.327} C_VEL
LIN {X 0,Y 219.346,Z 470.224,A -85,B 0,C 180,E1 -20633.358,E2 -20633.358} C_VEL
LIN {X 0,Y 221.806,Z 458.471,A -85,B 0,C 180,E1 -20635.324,E2 -20635.324} C_VEL
LIN {X 0,Y 223.823,Z 446.803,A -85,B 0,C 180,E1 -20636.83,E2 -20636.83} C_VEL
LIN {X 0,Y 225.48,Z 434.663,A -85,B 0,C 180,E1 -20637.999,E2 -20637.999} C_VEL
LIN {X 0,Y 226.899,Z 421.532,A -85,B 0,C 180,E1 -20638.88,E2 -20638.88} C_VEL
LIN {X 0,Y 227.551,Z 408.951,A -85,B 0,C 180,E1 -20639.422,E2 -20639.422} C_VEL
LIN {X 0,Y 228.436,Z 380.08,A -85,B 0,C 180,E1 -20640.304,E2 -20640.304} C_VEL
LIN {X 0,Y 225.499,Z 341.209,A -85,B 0,C 180,E1 -20642.028,E2 -20642.028} C_VEL
LIN {X 0,Y 222.34,Z 311.416,A -85,B 0,C 180,E1 -20643.529,E2 -20643.529} C_VEL
LIN {X 0,Y 219.562,Z 303.482,A -85,B 0,C 180,E1 -20644.305,E2 -20644.305} C_VEL
LIN {X 0,Y 217.123,Z 291.774,A -85,B 0,C 180,E1 -20648.34,E2 -20648.34} C_VEL
LIN {X 0,Y 214.239,Z 280.952,A -85,B 0,C 180,E1 -20652.43,E2 -20652.43} C_VEL
LIN {X 0,Y 213.704,Z 278.941,A -85,B 0,C 180,E1 -20653.313,E2 -20653.313} C_VEL
LIN {X 0,Y 213.696,Z 278.832,A -85,B 0,C 180,E1 -20656.344,E2 -20656.344} C_VEL
LIN {X 0,Y 213.7,Z 278.852,A -85,B 0,C 180,E1 -20661.329,E2 -20661.329} C_VEL
LIN {X 0,Y 213.749,Z 278.849,A -85,B 0,C 180,E1 -20666.017,E2 -20666.017} C_VEL
LIN {X 0,Y 213.742,Z 278.858,A -85,B 0,C 180,E1 -20670.448,E2 -20670.448} C_VEL
LIN {X 0,Y 213.772,Z 278.84,A -85,B 0,C 180,E1 -20674.698,E2 -20674.698} C_VEL
LIN {X 0,Y 213.77,Z 278.857,A -85,B 0,C 180,E1 -20678.799,E2 -20678.799} C_VEL
LIN {X 0,Y 213.875,Z 278.825,A -85,B 0,C 180,E1 -20682.798,E2 -20682.798} C_VEL
LIN {X 0,Y 213.925,Z 278.837,A -85,B 0,C 180,E1 -20686.705,E2 -20686.705} C_VEL
LIN {X 0,Y 214.125,Z 278.79,A -85,B 0,C 180,E1 -20690.555,E2 -20690.555} C_VEL
LIN {X 0,Y 214.065,Z 278.82,A -85,B 0,C 180,E1 -20694.348,E2 -20694.348} C_VEL
LIN {X 0,Y 214.396,Z 278.759,A -85,B 0,C 180,E1 -20698.122,E2 -20698.122} C_VEL
LIN {X 0,Y 214.501,Z 278.742,A -85,B 0,C 180,E1 -20700,E2 -20700} C_VEL
LIN {X 0,Y 214.392,Z 278.772,A -85,B 0,C 180,E1 -20701.879,E2 -20701.879} C_VEL
LIN {X 0,Y 214.162,Z 278.787,A -85,B 0,C 180,E1 -20707.543,E2 -20707.543} C_VEL
LIN {X 0,Y 213.979,Z 278.824,A -85,B 0,C 180,E1 -20711.366,E2 -20711.366} C_VEL
LIN {X 0,Y 213.89,Z 278.834,A -85,B 0,C 180,E1 -20715.241,E2 -20715.241} C_VEL
LIN {X 0,Y 213.788,Z 278.841,A -85,B 0,C 180,E1 -20719.193,E2 -20719.193} C_VEL
LIN {X 0,Y 213.778,Z 278.853,A -85,B 0,C 180,E1 -20723.236,E2 -20723.236} C_VEL
LIN {X 0,Y 213.761,Z 278.846,A -85,B 0,C 180,E1 -20727.418,E2 -20727.418} C_VEL
LIN {X 0,Y 213.753,Z 278.852,A -85,B 0,C 180,E1 -20731.741,E2 -20731.741} C_VEL
LIN {X 0,Y 213.737,Z 278.862,A -85,B 0,C 180,E1 -20736.29,E2 -20736.29} C_VEL
LIN {X 0,Y 213.692,Z 278.825,A -85,B 0,C 180,E1 -20741.131,E2 -20741.131} C_VEL
LIN {X 0,Y 213.698,Z 278.811,A -85,B 0,C 180,E1 -20743.682,E2 -20743.682} C_VEL
LIN {X 0,Y 213.698,Z 278.85,A -85,B 0,C 180,E1 -20746.347,E2 -20746.347} C_VEL
LIN {X 0,Y 213.7,Z 278.864,A -85,B 0,C 180,E1 -20749.149,E2 -20749.149} C_VEL
LIN {X 0,Y 213.74,Z 278.824,A -85,B 0,C 180,E1 -20753.713,E2 -20753.713} C_VEL
LIN {X 0,Y 213.758,Z 278.841,A -85,B 0,C 180,E1 -20758.263,E2 -20758.263} C_VEL
LIN {X 0,Y 213.842,Z 279.065,A -85,B 0,C 180,E1 -20763.462,E2 -20763.462} C_VEL
LIN {X 0,Y 214.052,Z 280.025,A -85,B 0,C 180,E1 -20763.773,E2 -20763.773} C_VEL
LIN {X 0,Y 224.05,Z 299.098,A -85,B 0,C 180,E1 -20766.055,E2 -20766.055} C_VEL
LIN {X 0,Y 230.526,Z 313.796,A -85,B 0,C 180,E1 -20767.468,E2 -20767.468} C_VEL
LIN {X 0,Y 229.21,Z 363.262,A -85,B 0,C 180,E1 -20769.027,E2 -20769.027} C_VEL
LIN {X 0,Y 228.562,Z 376.195,A -85,B 0,C 180,E1 -20769.69,E2 -20769.69} C_VEL
LIN {X 0,Y 227.8,Z 387.87,A -85,B 0,C 180,E1 -20770.632,E2 -20770.632} C_VEL
LIN {X 0,Y 226.437,Z 399.854,A -85,B 0,C 180,E1 -20771.92,E2 -20771.92} C_VEL
LIN {X 0,Y 224.817,Z 410.708,A -85,B 0,C 180,E1 -20773.427,E2 -20773.427} C_VEL
LIN {X 0,Y 222.963,Z 421.779,A -85,B 0,C 180,E1 -20775.395,E2 -20775.395} C_VEL
LIN {X 0,Y 221.103,Z 431.579,A -85,B 0,C 180,E1 -20777.612,E2 -20777.612} C_VEL
LIN {X 0,Y 219.012,Z 441.109,A -85,B 0,C 180,E1 -20780.302,E2 -20780.302} C_VEL
LIN {X 0,Y 217.255,Z 448.713,A -85,B 0,C 180,E1 -20783.033,E2 -20783.033} C_VEL
LIN {X 0,Y 215.698,Z 455.707,A -85,B 0,C 180,E1 -20786.265,E2 -20786.265} C_VEL
LIN {X 0,Y 214.72,Z 460.376,A -85,B 0,C 180,E1 -20789.063,E2 -20789.063} C_VEL
LIN {X 0,Y 213.922,Z 463.982,A -85,B 0,C 180,E1 -20791.883,E2 -20791.883} C_VEL
LIN {X 0,Y 213.691,Z 465.837,A -85,B 0,C 180,E1 -20793.772,E2 -20793.772} C_VEL
LIN {X 0,Y 213.681,Z 467.223,A -85,B 0,C 180,E1 -20795.663,E2 -20795.663} C_VEL
LIN {X 0,Y 213.778,Z 468.89,A -85,B 0,C 180,E1 -20799.505,E2 -20799.505} C_VEL
LIN {X 0,Y 214.018,Z 469.131,A -85,B 0,C 180,E1 -20801.364,E2 -20801.364} C_VEL
LIN {X 0,Y 214.973,Z 468.394,A -85,B 0,C 180,E1 -20805.162,E2 -20805.162} C_VEL
LIN {X 0,Y 215.697,Z 467.448,A -85,B 0,C 180,E1 -20807.053,E2 -20807.053} C_VEL
LIN {X 0,Y 217.513,Z 464.643,A -85,B 0,C 180,E1 -20810.442,E2 -20810.442} C_VEL
LIN {X 0,Y 219.585,Z 460.684,A -85,B 0,C 180,E1 -20813.583,E2 -20813.583} C_VEL
LIN {X 0,Y 221.853,Z 455.975,A -85,B 0,C 180,E1 -20816.328,E2 -20816.328} C_VEL
LIN {X 0,Y 224.499,Z 450.097,A -85,B 0,C 180,E1 -20818.969,E2 -20818.969} C_VEL
LIN {X 0,Y 227.583,Z 442.447,A -85,B 0,C 180,E1 -20821.667,E2 -20821.667} C_VEL
LIN {X 0,Y 230.905,Z 433.162,A -85,B 0,C 180,E1 -20824.19,E2 -20824.19} C_VEL
LIN {X 0,Y 234.024,Z 422.967,A -85,B 0,C 180,E1 -20826.378,E2 -20826.378} C_VEL
LIN {X 0,Y 236.577,Z 413.069,A -85,B 0,C 180,E1 -20828.055,E2 -20828.055} C_VEL
LIN {X 0,Y 238.906,Z 402.213,A -85,B 0,C 180,E1 -20829.505,E2 -20829.505} C_VEL
LIN {X 0,Y 240.816,Z 391.205,A -85,B 0,C 180,E1 -20830.642,E2 -20830.642} C_VEL
LIN {X 0,Y 242.16,Z 379.226,A -85,B 0,C 180,E1 -20831.599,E2 -20831.599} C_VEL
LIN {X 0,Y 243.011,Z 367.446,A -85,B 0,C 180,E1 -20832.248,E2 -20832.248} C_VEL
LIN {X 0,Y 244.185,Z 336.449,A -85,B 0,C 180,E1 -20833.231,E2 -20833.231} C_VEL
LIN {X 0,Y 244.408,Z 328.552,A -85,B 0,C 180,E1 -20833.484,E2 -20833.484} C_VEL
LIN {X 0,Y 236.631,Z 314.01,A -85,B 0,C 180,E1 -20835.651,E2 -20835.651} C_VEL
LIN {X 0,Y 228.519,Z 300.81,A -85,B 0,C 180,E1 -20838.075,E2 -20838.075} C_VEL
LIN {X 0,Y 222.344,Z 291.868,A -85,B 0,C 180,E1 -20840.068,E2 -20840.068} C_VEL
LIN {X 0,Y 219.591,Z 287.958,A -85,B 0,C 180,E1 -20841.016,E2 -20841.016} C_VEL
LIN {X 0,Y 217.392,Z 284.715,A -85,B 0,C 180,E1 -20841.808,E2 -20841.808} C_VEL
LIN {X 0,Y 216.467,Z 283.621,A -85,B 0,C 180,E1 -20842.137,E2 -20842.137} C_VEL
LIN {X 0,Y 214.564,Z 281.293,A -85,B 0,C 180,E1 -20842.832,E2 -20842.832} C_VEL
LIN {X 0,Y 213.861,Z 279.44,A -85,B 0,C 180,E1 -20843.282,E2 -20843.282} C_VEL
LIN {X 0,Y 213.741,Z 278.927,A -85,B 0,C 180,E1 -20843.71,E2 -20843.71} C_VEL
LIN {X 0,Y 213.758,Z 278.817,A -85,B 0,C 180,E1 -20848.26,E2 -20848.26} C_VEL
LIN {X 0,Y 213.785,Z 278.841,A -85,B 0,C 180,E1 -20852.597,E2 -20852.597} C_VEL
LIN {X 0,Y 213.81,Z 278.794,A -85,B 0,C 180,E1 -20856.979,E2 -20856.979} C_VEL
LIN {X 0,Y 213.942,Z 278.836,A -85,B 0,C 180,E1 -20862.803,E2 -20862.803} C_VEL
LIN {X 0,Y 213.95,Z 278.823,A -85,B 0,C 180,E1 -20866.706,E2 -20866.706} C_VEL
LIN {X 0,Y 214.131,Z 278.792,A -85,B 0,C 180,E1 -20870.554,E2 -20870.554} C_VEL
LIN {X 0,Y 214.068,Z 278.813,A -85,B 0,C 180,E1 -20874.347,E2 -20874.347} C_VEL
LIN {X 0,Y 214.401,Z 278.772,A -85,B 0,C 180,E1 -20878.121,E2 -20878.121} C_VEL
LIN {X 0,Y 214.509,Z 278.759,A -85,B 0,C 180,E1 -20880,E2 -20880} C_VEL
LIN {X 0,Y 214.403,Z 278.758,A -85,B 0,C 180,E1 -20881.878,E2 -20881.878} C_VEL
LIN {X 0,Y 214.174,Z 278.786,A -85,B 0,C 180,E1 -20887.542,E2 -20887.542} C_VEL
LIN {X 0,Y 213.99,Z 278.822,A -85,B 0,C 180,E1 -20891.364,E2 -20891.364} C_VEL
LIN {X 0,Y 213.906,Z 278.838,A -85,B 0,C 180,E1 -20895.239,E2 -20895.239} C_VEL
LIN {X 0,Y 213.819,Z 278.846,A -85,B 0,C 180,E1 -20899.189,E2 -20899.189} C_VEL
LIN {X 0,Y 213.8,Z 278.85,A -85,B 0,C 180,E1 -20903.232,E2 -20903.232} C_VEL
LIN {X 0,Y 213.783,Z 278.819,A -85,B 0,C 180,E1 -20907.427,E2 -20907.427} C_VEL
LIN {X 0,Y 213.757,Z 278.847,A -85,B 0,C 180,E1 -20911.739,E2 -20911.739} C_VEL
LIN {X 0,Y 213.773,Z 279.012,A -85,B 0,C 180,E1 -20915.9,E2 -20915.9} C_VEL
LIN {X 0,Y 216.224,Z 286.335,A -85,B 0,C 180,E1 -20919.936,E2 -20919.936} C_VEL
LIN {X 0,Y 218.604,Z 293.786,A -85,B 0,C 180,E1 -20923.608,E2 -20923.608} C_VEL
LIN {X 0,Y 219.132,Z 296.067,A -85,B 0,C 180,E1 -20924.426,E2 -20924.426} C_VEL
LIN {X 0,Y 219.805,Z 300.529,A -85,B 0,C 180,E1 -20925.419,E2 -20925.419} C_VEL
LIN {X 0,Y 220.484,Z 305.645,A -85,B 0,C 180,E1 -20926.198,E2 -20926.198} C_VEL
LIN {X 0,Y 222.281,Z 314.688,A -85,B 0,C 180,E1 -20927.328,E2 -20927.328} C_VEL
LIN {X 0,Y 224.225,Z 319.669,A -85,B 0,C 180,E1 -20928.072,E2 -20928.072} C_VEL
LIN {X 0,Y 229.589,Z 331.37,A -85,B 0,C 180,E1 -20929.872,E2 -20929.872} C_VEL
LIN {X 0,Y 231.3,Z 335.877,A -85,B 0,C 180,E1 -20930.45,E2 -20930.45} C_VEL
LIN {X 0,Y 234.305,Z 361.054,A -85,B 0,C 180,E1 -20932.122,E2 -20932.122} C_VEL
LIN {X 0,Y 236.253,Z 383.002,A -85,B 0,C 180,E1 -20933.379,E2 -20933.379} C_VEL
LIN {X 0,Y 236.024,Z 391.644,A -85,B 0,C 180,E1 -20933.667,E2 -20933.667} C_VEL
LIN {X 0,Y 234.682,Z 414.493,A -85,B 0,C 180,E1 -20934.373,E2 -20934.373} C_VEL
LIN {X 0,Y 233.11,Z 427.466,A -85,B 0,C 180,E1 -20935.052,E2 -20935.052} C_VEL
LIN {X 0,Y 230.908,Z 439.772,A -85,B 0,C 180,E1 -20935.995,E2 -20935.995} C_VEL
LIN {X 0,Y 227.883,Z 452.421,A -85,B 0,C 180,E1 -20937.336,E2 -20937.336} C_VEL
LIN {X 0,Y 224.449,Z 463.709,A -85,B 0,C 180,E1 -20938.892,E2 -20938.892} C_VEL
LIN {X 0,Y 220.896,Z 473.914,A -85,B 0,C 180,E1 -20940.714,E2 -20940.714} C_VEL
LIN {X 0,Y 217.186,Z 483.975,A -85,B 0,C 180,E1 -20943.062,E2 -20943.062} C_VEL
LIN {X 0,Y 213.599,Z 492.885,A -85,B 0,C 180,E1 -20945.714,E2 -20945.714} C_VEL
LIN {X 0,Y 210.714,Z 500.083,A -85,B 0,C 180,E1 -20948.476,E2 -20948.476} C_VEL
LIN {X 0,Y 208.338,Z 505.891,A -85,B 0,C 180,E1 -20951.308,E2 -20951.308} C_VEL
LIN {X 0,Y 206.742,Z 510.546,A -85,B 0,C 180,E1 -20954.219,E2 -20954.219} C_VEL
LIN {X 0,Y 205.589,Z 514.137,A -85,B 0,C 180,E1 -20957.161,E2 -20957.161} C_VEL
LIN {X 0,Y 205.095,Z 516.771,A -85,B 0,C 180,E1 -20960.134,E2 -20960.134} C_VEL
LIN {X 0,Y 205.314,Z 518.837,A -85,B 0,C 180,E1 -20964.105,E2 -20964.105} C_VEL
LIN {X 0,Y 205.636,Z 519.283,A -85,B 0,C 180,E1 -20966.08,E2 -20966.08} C_VEL
LIN {X 0,Y 205.957,Z 519.321,A -85,B 0,C 180,E1 -20968.044,E2 -20968.044} C_VEL
LIN {X 0,Y 206.109,Z 518.887,A -85,B 0,C 180,E1 -20969.999,E2 -20969.999} C_VEL
LIN {X 0,Y 206.03,Z 517.991,A -85,B 0,C 180,E1 -20971.954,E2 -20971.954} C_VEL
LIN {X 0,Y 205.768,Z 516.647,A -85,B 0,C 180,E1 -20973.916,E2 -20973.916} C_VEL
LIN {X 0,Y 205.369,Z 513.546,A -85,B 0,C 180,E1 -20977.061,E2 -20977.061} C_VEL
LIN {X 0,Y 205.267,Z 509.782,A -85,B 0,C 180,E1 -20979.856,E2 -20979.856} C_VEL
LIN {X 0,Y 205.702,Z 504.67,A -85,B 0,C 180,E1 -20982.83,E2 -20982.83} C_VEL
LIN {X 0,Y 206.627,Z 498.252,A -85,B 0,C 180,E1 -20985.788,E2 -20985.788} C_VEL
LIN {X 0,Y 207.838,Z 491.486,A -85,B 0,C 180,E1 -20988.305,E2 -20988.305} C_VEL
LIN {X 0,Y 209.506,Z 483.884,A -85,B 0,C 180,E1 -20990.622,E2 -20990.622} C_VEL
LIN {X 0,Y 211.699,Z 474.405,A -85,B 0,C 180,E1 -20992.958,E2 -20992.958} C_VEL
LIN {X 0,Y 213.589,Z 465.149,A -85,B 0,C 180,E1 -20994.803,E2 -20994.803} C_VEL
LIN {X 0,Y 215.6,Z 455.36,A -85,B 0,C 180,E1 -20996.367,E2 -20996.367} C_VEL
LIN {X 0,Y 217.822,Z 442.978,A -85,B 0,C 180,E1 -20997.893,E2 -20997.893} C_VEL
LIN {X 0,Y 219.538,Z 429.927,A -85,B 0,C 180,E1 -20999.082,E2 -20999.082} C_VEL
LIN {X 0,Y 220.722,Z 416.866,A -85,B 0,C 180,E1 -20999.876,E2 -20999.876} C_VEL
LIN {X 0,Y 221.592,Z 396.772,A -85,B 0,C 180,E1 -21000.578,E2 -21000.578} C_VEL
LIN {X 0,Y 222.023,Z 380.249,A -85,B 0,C 180,E1 -21001.108,E2 -21001.108} C_VEL
LIN {X 0,Y 219.32,Z 342.873,A -85,B 0,C 180,E1 -21002.822,E2 -21002.822} C_VEL
LIN {X 0,Y 216.301,Z 313.463,A -85,B 0,C 180,E1 -21004.355,E2 -21004.355} C_VEL
LIN {X 0,Y 212.225,Z 302.563,A -85,B 0,C 180,E1 -21005.469,E2 -21005.469} C_VEL
LIN {X 0,Y 210.123,Z 292.871,A -85,B 0,C 180,E1 -21008.956,E2 -21008.956} C_VEL
LIN {X 0,Y 207.684,Z 283.583,A -85,B 0,C 180,E1 -21012.592,E2 -21012.592} C_VEL
LIN {X 0,Y 206.627,Z 279.824,A -85,B 0,C 180,E1 -21014.234,E2 -21014.234} C_VEL
LIN {X 0,Y 206.625,Z 279.745,A -85,B 0,C 180,E1 -21018.44,E2 -21018.44} C_VEL
LIN {X 0,Y 206.666,Z 279.729,A -85,B 0,C 180,E1 -21022.258,E2 -21022.258} C_VEL
LIN {X 0,Y 206.688,Z 279.718,A -85,B 0,C 180,E1 -21027.041,E2 -21027.041} C_VEL
LIN {X 0,Y 206.701,Z 279.737,A -85,B 0,C 180,E1 -21032.127,E2 -21032.127} C_VEL
LIN {X 0,Y 206.731,Z 279.727,A -85,B 0,C 180,E1 -21036.614,E2 -21036.614} C_VEL
LIN {X 0,Y 206.796,Z 279.704,A -85,B 0,C 180,E1 -21042.19,E2 -21042.19} C_VEL
LIN {X 0,Y 206.865,Z 279.717,A -85,B 0,C 180,E1 -21046.243,E2 -21046.243} C_VEL
LIN {X 0,Y 207.07,Z 279.668,A -85,B 0,C 180,E1 -21050.23,E2 -21050.23} C_VEL
LIN {X 0,Y 207.029,Z 279.695,A -85,B 0,C 180,E1 -21054.155,E2 -21054.155} C_VEL
LIN {X 0,Y 207.336,Z 279.638,A -85,B 0,C 180,E1 -21058.058,E2 -21058.058} C_VEL
LIN {X 0,Y 207.47,Z 279.617,A -85,B 0,C 180,E1 -21060,E2 -21060} C_VEL
LIN {X 0,Y 207.332,Z 279.651,A -85,B 0,C 180,E1 -21061.943,E2 -21061.943} C_VEL
LIN {X 0,Y 207.108,Z 279.663,A -85,B 0,C 180,E1 -21067.802,E2 -21067.802} C_VEL
LIN {X 0,Y 206.903,Z 279.707,A -85,B 0,C 180,E1 -21071.76,E2 -21071.76} C_VEL
LIN {X 0,Y 206.817,Z 279.707,A -85,B 0,C 180,E1 -21075.775,E2 -21075.775} C_VEL
LIN {X 0,Y 206.708,Z 279.727,A -85,B 0,C 180,E1 -21079.877,E2 -21079.877} C_VEL
LIN {X 0,Y 206.691,Z 279.727,A -85,B 0,C 180,E1 -21084.082,E2 -21084.082} C_VEL
LIN {X 0,Y 206.673,Z 279.736,A -85,B 0,C 180,E1 -21088.43,E2 -21088.43} C_VEL
LIN {X 0,Y 206.689,Z 279.722,A -85,B 0,C 180,E1 -21092.96,E2 -21092.96} C_VEL
LIN {X 0,Y 206.664,Z 279.741,A -85,B 0,C 180,E1 -21097.744,E2 -21097.744} C_VEL
LIN {X 0,Y 206.626,Z 279.697,A -85,B 0,C 180,E1 -21101.56,E2 -21101.56} C_VEL
LIN {X 0,Y 206.626,Z 279.713,A -85,B 0,C 180,E1 -21105.585,E2 -21105.585} C_VEL
LIN {X 0,Y 206.644,Z 279.737,A -85,B 0,C 180,E1 -21109.747,E2 -21109.747} C_VEL
LIN {X 0,Y 206.698,Z 279.71,A -85,B 0,C 180,E1 -21114.69,E2 -21114.69} C_VEL
LIN {X 0,Y 206.693,Z 279.711,A -85,B 0,C 180,E1 -21119.336,E2 -21119.336} C_VEL
LIN {X 0,Y 206.744,Z 279.917,A -85,B 0,C 180,E1 -21122.226,E2 -21122.226} C_VEL
LIN {X 0,Y 206.975,Z 280.86,A -85,B 0,C 180,E1 -21122.587,E2 -21122.587} C_VEL
LIN {X 0,Y 208.555,Z 283.64,A -85,B 0,C 180,E1 -21123.012,E2 -21123.012} C_VEL
LIN {X 0,Y 218.461,Z 302.479,A -85,B 0,C 180,E1 -21125.352,E2 -21125.352} C_VEL
LIN {X 0,Y 224.227,Z 315.594,A -85,B 0,C 180,E1 -21126.674,E2 -21126.674} C_VEL
LIN {X 0,Y 222.875,Z 364.168,A -85,B 0,C 180,E1 -21128.249,E2 -21128.249} C_VEL
LIN {X 0,Y 222.21,Z 377.174,A -85,B 0,C 180,E1 -21128.938,E2 -21128.938} C_VEL
LIN {X 0,Y 221.237,Z 390.135,A -85,B 0,C 180,E1 -21130.033,E2 -21130.033} C_VEL
LIN {X 0,Y 219.785,Z 401.819,A -85,B 0,C 180,E1 -21131.352,E2 -21131.352} C_VEL
LIN {X 0,Y 218.122,Z 412.453,A -85,B 0,C 180,E1 -21132.903,E2 -21132.903} C_VEL
LIN {X 0,Y 216.198,Z 423.299,A -85,B 0,C 180,E1 -21134.928,E2 -21134.928} C_VEL
LIN {X 0,Y 214.253,Z 432.99,A -85,B 0,C 180,E1 -21137.209,E2 -21137.209} C_VEL
LIN {X 0,Y 212.447,Z 440.957,A -85,B 0,C 180,E1 -21139.518,E2 -21139.518} C_VEL
LIN {X 0,Y 210.587,Z 448.79,A -85,B 0,C 180,E1 -21142.329,E2 -21142.329} C_VEL
LIN {X 0,Y 209.154,Z 455.042,A -85,B 0,C 180,E1 -21145.182,E2 -21145.182} C_VEL
LIN {X 0,Y 208.012,Z 460.031,A -85,B 0,C 180,E1 -21148.065,E2 -21148.065} C_VEL
LIN {X 0,Y 207.089,Z 463.933,A -85,B 0,C 180,E1 -21150.973,E2 -21150.973} C_VEL
LIN {X 0,Y 206.634,Z 466.81,A -85,B 0,C 180,E1 -21153.901,E2 -21153.901} C_VEL
LIN {X 0,Y 206.617,Z 468.167,A -85,B 0,C 180,E1 -21155.858,E2 -21155.858} C_VEL
LIN {X 0,Y 206.774,Z 469.77,A -85,B 0,C 180,E1 -21159.785,E2 -21159.785} C_VEL
LIN {X 0,Y 207.037,Z 469.977,A -85,B 0,C 180,E1 -21161.752,E2 -21161.752} C_VEL
LIN {X 0,Y 208.091,Z 469.187,A -85,B 0,C 180,E1 -21165.676,E2 -21165.676} C_VEL
LIN {X 0,Y 208.877,Z 468.215,A -85,B 0,C 180,E1 -21167.627,E2 -21167.627} C_VEL
LIN {X 0,Y 210.704,Z 465.526,A -85,B 0,C 180,E1 -21170.941,E2 -21170.941} C_VEL
LIN {X 0,Y 213.038,Z 461.314,A -85,B 0,C 180,E1 -21174.354,E2 -21174.354} C_VEL
LIN {X 0,Y 215.457,Z 456.544,A -85,B 0,C 180,E1 -21177.172,E2 -21177.172} C_VEL
LIN {X 0,Y 218.314,Z 450.474,A -85,B 0,C 180,E1 -21179.932,E2 -21179.932} C_VEL
LIN {X 0,Y 221.519,Z 442.841,A -85,B 0,C 180,E1 -21182.639,E2 -21182.639} C_VEL
LIN {X 0,Y 224.907,Z 433.737,A -85,B 0,C 180,E1 -21185.145,E2 -21185.145} C_VEL
LIN {X 0,Y 227.948,Z 424.206,A -85,B 0,C 180,E1 -21187.234,E2 -21187.234} C_VEL
LIN {X 0,Y 230.613,Z 414.426,A -85,B 0,C 180,E1 -21188.943,E2 -21188.943} C_VEL
LIN {X 0,Y 233.036,Z 403.71,A -85,B 0,C 180,E1 -21190.421,E2 -21190.421} C_VEL
LIN {X 0,Y 235.163,Z 392.022,A -85,B 0,C 180,E1 -21191.656,E2 -21191.656} C_VEL
LIN {X 0,Y 236.553,Z 380.33,A -85,B 0,C 180,E1 -21192.608,E2 -21192.608} C_VEL
LIN {X 0,Y 237.512,Z 367.769,A -85,B 0,C 180,E1 -21193.31,E2 -21193.31} C_VEL
LIN {X 0,Y 238.917,Z 331.039,A -85,B 0,C 180,E1 -21194.492,E2 -21194.492} C_VEL
LIN {X 0,Y 231.447,Z 317.25,A -85,B 0,C 180,E1 -21196.68,E2 -21196.68} C_VEL
LIN {X 0,Y 224.347,Z 305.607,A -85,B 0,C 180,E1 -21198.914,E2 -21198.914} C_VEL
LIN {X 0,Y 218.522,Z 296.969,A -85,B 0,C 180,E1 -21200.891,E2 -21200.891} C_VEL
LIN {X 0,Y 215.67,Z 292.958,A -85,B 0,C 180,E1 -21201.915,E2 -21201.915} C_VEL
LIN {X 0,Y 212.992,Z 289.16,A -85,B 0,C 180,E1 -21202.924,E2 -21202.924} C_VEL
LIN {X 0,Y 210.898,Z 286.382,A -85,B 0,C 180,E1 -21203.735,E2 -21203.735} C_VEL
LIN {X 0,Y 210.186,Z 285.061,A -85,B 0,C 180,E1 -21204.038,E2 -21204.038} C_VEL
LIN {X 0,Y 207.905,Z 282.902,A -85,B 0,C 180,E1 -21204.923,E2 -21204.923} C_VEL
LIN {X 0,Y 206.809,Z 280.314,A -85,B 0,C 180,E1 -21205.599,E2 -21205.599} C_VEL
LIN {X 0,Y 206.719,Z 279.785,A -85,B 0,C 180,E1 -21206.17,E2 -21206.17} C_VEL
LIN {X 0,Y 206.695,Z 279.688,A -85,B 0,C 180,E1 -21209.334,E2 -21209.334} C_VEL
LIN {X 0,Y 206.705,Z 279.741,A -85,B 0,C 180,E1 -21213.768,E2 -21213.768} C_VEL
LIN {X 0,Y 206.734,Z 279.668,A -85,B 0,C 180,E1 -21218.04,E2 -21218.04} C_VEL
LIN {X 0,Y 206.872,Z 279.711,A -85,B 0,C 180,E1 -21222.196,E2 -21222.196} C_VEL
LIN {X 0,Y 206.892,Z 279.698,A -85,B 0,C 180,E1 -21226.244,E2 -21226.244} C_VEL
LIN {X 0,Y 207.076,Z 279.671,A -85,B 0,C 180,E1 -21230.229,E2 -21230.229} C_VEL
LIN {X 0,Y 207.032,Z 279.692,A -85,B 0,C 180,E1 -21234.154,E2 -21234.154} C_VEL
LIN {X 0,Y 207.34,Z 279.651,A -85,B 0,C 180,E1 -21238.057,E2 -21238.057} C_VEL
LIN {X 0,Y 207.477,Z 279.634,A -85,B 0,C 180,E1 -21240,E2 -21240} C_VEL
LIN {X 0,Y 207.342,Z 279.637,A -85,B 0,C 180,E1 -21241.942,E2 -21241.942} C_VEL
LIN {X 0,Y 207.118,Z 279.665,A -85,B 0,C 180,E1 -21247.8,E2 -21247.8} C_VEL
LIN {X 0,Y 206.913,Z 279.698,A -85,B 0,C 180,E1 -21251.759,E2 -21251.759} C_VEL
LIN {X 0,Y 206.841,Z 279.721,A -85,B 0,C 180,E1 -21255.772,E2 -21255.772} C_VEL
LIN {X 0,Y 206.856,Z 279.707,A -85,B 0,C 180,E1 -21257.954,E2 -21257.954} C_VEL
LIN {X 0,Y 206.743,Z 279.73,A -85,B 0,C 180,E1 -21263.39,E2 -21263.39} C_VEL
LIN {X 0,Y 206.685,Z 279.706,A -85,B 0,C 180,E1 -21268.427,E2 -21268.427} C_VEL
LIN {X 0,Y 206.693,Z 279.713,A -85,B 0,C 180,E1 -21272.958,E2 -21272.958} C_VEL
LIN {X 0,Y 206.745,Z 279.907,A -85,B 0,C 180,E1 -21273.97,E2 -21273.97} C_VEL
LIN {X 0,Y 209.093,Z 286.744,A -85,B 0,C 180,E1 -21278.056,E2 -21278.056} C_VEL
LIN {X 0,Y 211.812,Z 295.15,A -85,B 0,C 180,E1 -21282.479,E2 -21282.479} C_VEL
LIN {X 0,Y 212.714,Z 298.061,A -85,B 0,C 180,E1 -21283.775,E2 -21283.775} C_VEL
LIN {X 0,Y 219.915,Z 311.085,A -85,B 0,C 180,E1 -21286.555,E2 -21286.555} C_VEL
LIN {X 0,Y 224.225,Z 319.669,A -85,B 0,C 180,E1 -21288.072,E2 -21288.072} C_VEL
LIN {X 0,Y 225.528,Z 322.898,A -85,B 0,C 180,E1 -21288.539,E2 -21288.539} C_VEL
LIN {X 0,Y 226.669,Z 328.357,A -85,B 0,C 180,E1 -21289.054,E2 -21289.054} C_VEL
LIN {X 0,Y 227.117,Z 334.158,A -85,B 0,C 180,E1 -21289.41,E2 -21289.41} C_VEL
LIN {X 0,Y 227.648,Z 350.28,A -85,B 0,C 180,E1 -21290.219,E2 -21290.219} C_VEL
LIN {X 0,Y 230.258,Z 376.8,A -85,B 0,C 180,E1 -21291.895,E2 -21291.895} C_VEL
LIN {X 0,Y 230.846,Z 386.489,A -85,B 0,C 180,E1 -21292.411,E2 -21292.411} C_VEL
LIN {X 0,Y 229.329,Z 412.645,A -85,B 0,C 180,E1 -21293.213,E2 -21293.213} C_VEL
LIN {X 0,Y 227.623,Z 426.216,A -85,B 0,C 180,E1 -21293.91,E2 -21293.91} C_VEL
LIN {X 0,Y 225.549,Z 437.808,A -85,B 0,C 180,E1 -21294.799,E2 -21294.799} C_VEL
LIN {X 0,Y 222.852,Z 449.167,A -85,B 0,C 180,E1 -21295.96,E2 -21295.96} C_VEL
LIN {X 0,Y 219.243,Z 460.895,A -85,B 0,C 180,E1 -21297.525,E2 -21297.525} C_VEL
LIN {X 0,Y 215.529,Z 471.462,A -85,B 0,C 180,E1 -21299.369,E2 -21299.369} C_VEL
LIN {X 0,Y 212.191,Z 480.134,A -85,B 0,C 180,E1 -21301.298,E2 -21301.298} C_VEL
LIN {X 0,Y 208.898,Z 488.169,A -85,B 0,C 180,E1 -21303.527,E2 -21303.527} C_VEL
LIN {X 0,Y 205.478,Z 496.094,A -85,B 0,C 180,E1 -21306.304,E2 -21306.304} C_VEL
LIN {X 0,Y 202.353,Z 503.438,A -85,B 0,C 180,E1 -21309.676,E2 -21309.676} C_VEL
LIN {X 0,Y 200.369,Z 508.415,A -85,B 0,C 180,E1 -21312.654,E2 -21312.654} C_VEL
LIN {X 0,Y 198.945,Z 512.298,A -85,B 0,C 180,E1 -21315.683,E2 -21315.683} C_VEL
LIN {X 0,Y 198.363,Z 514.351,A -85,B 0,C 180,E1 -21317.726,E2 -21317.726} C_VEL
LIN {X 0,Y 198.058,Z 515.983,A -85,B 0,C 180,E1 -21319.78,E2 -21319.78} C_VEL
LIN {X 0,Y 198.241,Z 518.009,A -85,B 0,C 180,E1 -21323.894,E2 -21323.894} C_VEL
LIN {X 0,Y 198.545,Z 518.436,A -85,B 0,C 180,E1 -21325.94,E2 -21325.94} C_VEL
LIN {X 0,Y 198.901,Z 518.453,A -85,B 0,C 180,E1 -21327.974,E2 -21327.974} C_VEL
LIN {X 0,Y 199.061,Z 517.99,A -85,B 0,C 180,E1 -21329.999,E2 -21329.999} C_VEL
LIN {X 0,Y 198.975,Z 517.074,A -85,B 0,C 180,E1 -21332.023,E2 -21332.023} C_VEL
LIN {X 0,Y 198.673,Z 515.703,A -85,B 0,C 180,E1 -21334.056,E2 -21334.056} C_VEL
LIN {X 0,Y 198.29,Z 512.827,A -85,B 0,C 180,E1 -21337.067,E2 -21337.067} C_VEL
LIN {X 0,Y 198.232,Z 508.75,A -85,B 0,C 180,E1 -21340.21,E2 -21340.21} C_VEL
LIN {X 0,Y 198.836,Z 502.609,A -85,B 0,C 180,E1 -21343.802,E2 -21343.802} C_VEL
LIN {X 0,Y 199.898,Z 495.853,A -85,B 0,C 180,E1 -21346.86,E2 -21346.86} C_VEL
LIN {X 0,Y 201.749,Z 487.515,A -85,B 0,C 180,E1 -21349.856,E2 -21349.856} C_VEL
LIN {X 0,Y 203.682,Z 479.009,A -85,B 0,C 180,E1 -21352.305,E2 -21352.305} C_VEL
LIN {X 0,Y 205.771,Z 469.728,A -85,B 0,C 180,E1 -21354.463,E2 -21354.463} C_VEL
LIN {X 0,Y 208.153,Z 459.703,A -85,B 0,C 180,E1 -21356.303,E2 -21356.303} C_VEL
LIN {X 0,Y 210.2,Z 448.745,A -85,B 0,C 180,E1 -21357.909,E2 -21357.909} C_VEL
LIN {X 0,Y 212.177,Z 436.693,A -85,B 0,C 180,E1 -21359.245,E2 -21359.245} C_VEL
LIN {X 0,Y 213.804,Z 423.81,A -85,B 0,C 180,E1 -21360.271,E2 -21360.271} C_VEL
LIN {X 0,Y 214.674,Z 411.336,A -85,B 0,C 180,E1 -21360.928,E2 -21360.928} C_VEL
LIN {X 0,Y 215.701,Z 380.93,A -85,B 0,C 180,E1 -21361.934,E2 -21361.934} C_VEL
LIN {X 0,Y 213.1,Z 343.702,A -85,B 0,C 180,E1 -21363.704,E2 -21363.704} C_VEL
LIN {X 0,Y 210.247,Z 315.49,A -85,B 0,C 180,E1 -21365.238,E2 -21365.238} C_VEL
LIN {X 0,Y 204.876,Z 301.625,A -85,B 0,C 180,E1 -21366.741,E2 -21366.741} C_VEL
LIN {X 0,Y 203,Z 293.498,A -85,B 0,C 180,E1 -21369.8,E2 -21369.8} C_VEL
LIN {X 0,Y 200.397,Z 283.563,A -85,B 0,C 180,E1 -21373.885,E2 -21373.885} C_VEL
LIN {X 0,Y 199.59,Z 280.7,A -85,B 0,C 180,E1 -21375.232,E2 -21375.232} C_VEL
LIN {X 0,Y 199.564,Z 280.615,A -85,B 0,C 180,E1 -21378.001,E2 -21378.001} C_VEL
LIN {X 0,Y 199.592,Z 280.61,A -85,B 0,C 180,E1 -21380.771,E2 -21380.771} C_VEL
LIN {X 0,Y 199.607,Z 280.621,A -85,B 0,C 180,E1 -21384.074,E2 -21384.074} C_VEL
LIN {X 0,Y 199.679,Z 280.59,A -85,B 0,C 180,E1 -21388.133,E2 -21388.133} C_VEL
LIN {X 0,Y 199.634,Z 280.611,A -85,B 0,C 180,E1 -21392.764,E2 -21392.764} C_VEL
LIN {X 0,Y 199.671,Z 280.611,A -85,B 0,C 180,E1 -21397.221,E2 -21397.221} C_VEL
LIN {X 0,Y 199.738,Z 280.582,A -85,B 0,C 180,E1 -21401.803,E2 -21401.803} C_VEL
LIN {X 0,Y 199.803,Z 280.596,A -85,B 0,C 180,E1 -21405.746,E2 -21405.746} C_VEL
LIN {X 0,Y 200.016,Z 280.546,A -85,B 0,C 180,E1 -21409.882,E2 -21409.882} C_VEL
LIN {X 0,Y 199.992,Z 280.571,A -85,B 0,C 180,E1 -21413.949,E2 -21413.949} C_VEL
LIN {X 0,Y 200.278,Z 280.516,A -85,B 0,C 180,E1 -21417.989,E2 -21417.989} C_VEL
LIN {X 0,Y 200.437,Z 280.492,A -85,B 0,C 180,E1 -21420,E2 -21420} C_VEL
LIN {X 0,Y 199.971,Z 280.576,A -85,B 0,C 180,E1 -21424.031,E2 -21424.031} C_VEL
LIN {X 0,Y 200.057,Z 280.538,A -85,B 0,C 180,E1 -21428.078,E2 -21428.078} C_VEL
LIN {X 0,Y 199.854,Z 280.586,A -85,B 0,C 180,E1 -21432.181,E2 -21432.181} C_VEL
LIN {X 0,Y 199.755,Z 280.58,A -85,B 0,C 180,E1 -21436.348,E2 -21436.348} C_VEL
LIN {X 0,Y 199.64,Z 280.613,A -85,B 0,C 180,E1 -21440.612,E2 -21440.612} C_VEL
LIN {X 0,Y 199.613,Z 280.601,A -85,B 0,C 180,E1 -21444.993,E2 -21444.993} C_VEL
LIN {X 0,Y 199.598,Z 280.622,A -85,B 0,C 180,E1 -21449.535,E2 -21449.535} C_VEL
LIN {X 0,Y 199.66,Z 280.601,A -85,B 0,C 180,E1 -21452.354,E2 -21452.354} C_VEL
LIN {X 0,Y 199.613,Z 280.621,A -85,B 0,C 180,E1 -21456.766,E2 -21456.766} C_VEL
LIN {X 0,Y 199.59,Z 280.607,A -85,B 0,C 180,E1 -21459.333,E2 -21459.333} C_VEL
LIN {X 0,Y 199.561,Z 280.567,A -85,B 0,C 180,E1 -21462.308,E2 -21462.308} C_VEL
LIN {X 0,Y 199.572,Z 280.582,A -85,B 0,C 180,E1 -21465.229,E2 -21465.229} C_VEL
LIN {X 0,Y 199.568,Z 280.627,A -85,B 0,C 180,E1 -21468.004,E2 -21468.004} C_VEL
LIN {X 0,Y 199.594,Z 280.595,A -85,B 0,C 180,E1 -21470.775,E2 -21470.775} C_VEL
LIN {X 0,Y 199.61,Z 280.61,A -85,B 0,C 180,E1 -21475.715,E2 -21475.715} C_VEL
LIN {X 0,Y 199.685,Z 280.592,A -85,B 0,C 180,E1 -21478.136,E2 -21478.136} C_VEL
LIN {X 0,Y 199.651,Z 280.839,A -85,B 0,C 180,E1 -21480.988,E2 -21480.988} C_VEL
LIN {X 0,Y 199.988,Z 282.049,A -85,B 0,C 180,E1 -21481.36,E2 -21481.36} C_VEL
LIN {X 0,Y 206.321,Z 293.267,A -85,B 0,C 180,E1 -21483.009,E2 -21483.009} C_VEL
LIN {X 0,Y 214.212,Z 308.803,A -85,B 0,C 180,E1 -21484.934,E2 -21484.934} C_VEL
LIN {X 0,Y 217.965,Z 317.551,A -85,B 0,C 180,E1 -21485.84,E2 -21485.84} C_VEL
LIN {X 0,Y 216.555,Z 366.207,A -85,B 0,C 180,E1 -21487.47,E2 -21487.47} C_VEL
LIN {X 0,Y 215.9,Z 377.96,A -85,B 0,C 180,E1 -21488.127,E2 -21488.127} C_VEL
LIN {X 0,Y 214.932,Z 390.182,A -85,B 0,C 180,E1 -21489.171,E2 -21489.171} C_VEL
LIN {X 0,Y 213.427,Z 402.034,A -85,B 0,C 180,E1 -21490.526,E2 -21490.526} C_VEL
LIN {X 0,Y 211.68,Z 412.791,A -85,B 0,C 180,E1 -21492.116,E2 -21492.116} C_VEL
LIN {X 0,Y 209.664,Z 423.762,A -85,B 0,C 180,E1 -21494.197,E2 -21494.197} C_VEL
LIN {X 0,Y 207.427,Z 434.393,A -85,B 0,C 180,E1 -21496.78,E2 -21496.78} C_VEL
LIN {X 0,Y 205.519,Z 442.275,A -85,B 0,C 180,E1 -21499.16,E2 -21499.16} C_VEL
LIN {X 0,Y 203.608,Z 450.005,A -85,B 0,C 180,E1 -21502.065,E2 -21502.065} C_VEL
LIN {X 0,Y 202.121,Z 456.176,A -85,B 0,C 180,E1 -21505.014,E2 -21505.014} C_VEL
LIN {X 0,Y 200.945,Z 461.106,A -85,B 0,C 180,E1 -21507.997,E2 -21507.997} C_VEL
LIN {X 0,Y 200.016,Z 464.951,A -85,B 0,C 180,E1 -21511.007,E2 -21511.007} C_VEL
LIN {X 0,Y 199.579,Z 467.774,A -85,B 0,C 180,E1 -21514.039,E2 -21514.039} C_VEL
LIN {X 0,Y 199.558,Z 469.109,A -85,B 0,C 180,E1 -21516.066,E2 -21516.066} C_VEL
LIN {X 0,Y 199.765,Z 470.659,A -85,B 0,C 180,E1 -21520.132,E2 -21520.132} C_VEL
LIN {X 0,Y 200.572,Z 470.589,A -85,B 0,C 180,E1 -21524.199,E2 -21524.199} C_VEL
LIN {X 0,Y 202.079,Z 468.975,A -85,B 0,C 180,E1 -21528.241,E2 -21528.241} C_VEL
LIN {X 0,Y 203.942,Z 466.385,A -85,B 0,C 180,E1 -21531.494,E2 -21531.494} C_VEL
LIN {X 0,Y 206.542,Z 461.945,A -85,B 0,C 180,E1 -21535.172,E2 -21535.172} C_VEL
LIN {X 0,Y 209.108,Z 457.113,A -85,B 0,C 180,E1 -21538.069,E2 -21538.069} C_VEL
LIN {X 0,Y 212.02,Z 451.195,A -85,B 0,C 180,E1 -21540.806,E2 -21540.806} C_VEL
LIN {X 0,Y 214.919,Z 444.646,A -85,B 0,C 180,E1 -21543.212,E2 -21543.212} C_VEL
LIN {X 0,Y 218.027,Z 436.995,A -85,B 0,C 180,E1 -21545.466,E2 -21545.466} C_VEL
LIN {X 0,Y 221.241,Z 427.589,A -85,B 0,C 180,E1 -21547.698,E2 -21547.698} C_VEL
LIN {X 0,Y 224.378,Z 417.056,A -85,B 0,C 180,E1 -21549.657,E2 -21549.657} C_VEL
LIN {X 0,Y 226.858,Z 406.84,A -85,B 0,C 180,E1 -21551.172,E2 -21551.172} C_VEL
LIN {X 0,Y 229.337,Z 394.294,A -85,B 0,C 180,E1 -21552.587,E2 -21552.587} C_VEL
LIN {X 0,Y 230.989,Z 382.149,A -85,B 0,C 180,E1 -21553.605,E2 -21553.605} C_VEL
LIN {X 0,Y 231.794,Z 372.438,A -85,B 0,C 180,E1 -21554.215,E2 -21554.215} C_VEL
LIN {X 0,Y 232.511,Z 357.275,A -85,B 0,C 180,E1 -21554.803,E2 -21554.803} C_VEL
LIN {X 0,Y 233.41,Z 333.547,A -85,B 0,C 180,E1 -21555.567,E2 -21555.567} C_VEL
LIN {X 0,Y 226.256,Z 320.191,A -85,B 0,C 180,E1 -21557.792,E2 -21557.792} C_VEL
LIN {X 0,Y 219.909,Z 309.875,A -85,B 0,C 180,E1 -21559.897,E2 -21559.897} C_VEL
LIN {X 0,Y 212.678,Z 299.015,A -85,B 0,C 180,E1 -21562.522,E2 -21562.522} C_VEL
LIN {X 0,Y 209.322,Z 294.427,A -85,B 0,C 180,E1 -21563.829,E2 -21563.829} C_VEL
LIN {X 0,Y 206.797,Z 290.817,A -85,B 0,C 180,E1 -21564.874,E2 -21564.874} C_VEL
LIN {X 0,Y 204.313,Z 287.898,A -85,B 0,C 180,E1 -21565.918,E2 -21565.918} C_VEL
LIN {X 0,Y 203.272,Z 285.949,A -85,B 0,C 180,E1 -21566.413,E2 -21566.413} C_VEL
LIN {X 0,Y 200.974,Z 283.889,A -85,B 0,C 180,E1 -21567.412,E2 -21567.412} C_VEL
LIN {X 0,Y 199.804,Z 281.304,A -85,B 0,C 180,E1 -21568.155,E2 -21568.155} C_VEL
LIN {X 0,Y 199.685,Z 280.678,A -85,B 0,C 180,E1 -21568.725,E2 -21568.725} C_VEL
LIN {X 0,Y 199.642,Z 280.602,A -85,B 0,C 180,E1 -21572.764,E2 -21572.764} C_VEL
LIN {X 0,Y 199.707,Z 280.546,A -85,B 0,C 180,E1 -21577.225,E2 -21577.225} C_VEL
LIN {X 0,Y 199.795,Z 280.579,A -85,B 0,C 180,E1 -21581.758,E2 -21581.758} C_VEL
LIN {X 0,Y 199.833,Z 280.575,A -85,B 0,C 180,E1 -21585.748,E2 -21585.748} C_VEL
LIN {X 0,Y 200.022,Z 280.551,A -85,B 0,C 180,E1 -21589.881,E2 -21589.881} C_VEL
LIN {X 0,Y 199.996,Z 280.57,A -85,B 0,C 180,E1 -21593.948,E2 -21593.948} C_VEL
LIN {X 0,Y 200.282,Z 280.528,A -85,B 0,C 180,E1 -21597.989,E2 -21597.989} C_VEL
LIN {X 0,Y 200.444,Z 280.509,A -85,B 0,C 180,E1 -21600,E2 -21600} C_VEL
LIN {X 0,Y 199.989,Z 280.569,A -85,B 0,C 180,E1 -21604.03,E2 -21604.03} C_VEL
LIN {X 0,Y 200.067,Z 280.543,A -85,B 0,C 180,E1 -21608.077,E2 -21608.077} C_VEL
LIN {X 0,Y 199.864,Z 280.572,A -85,B 0,C 180,E1 -21612.18,E2 -21612.18} C_VEL
LIN {X 0,Y 199.786,Z 280.597,A -85,B 0,C 180,E1 -21616.345,E2 -21616.345} C_VEL
LIN {X 0,Y 199.673,Z 280.611,A -85,B 0,C 180,E1 -21620.608,E2 -21620.608} C_VEL
LIN {X 0,Y 199.647,Z 280.603,A -85,B 0,C 180,E1 -21624.987,E2 -21624.987} C_VEL
LIN {X 0,Y 199.606,Z 280.599,A -85,B 0,C 180,E1 -21629.533,E2 -21629.533} C_VEL
LIN {X 0,Y 199.709,Z 280.896,A -85,B 0,C 180,E1 -21631.861,E2 -21631.861} C_VEL
LIN {X 0,Y 201.45,Z 285.859,A -85,B 0,C 180,E1 -21635.144,E2 -21635.144} C_VEL
LIN {X 0,Y 203.375,Z 291.414,A -85,B 0,C 180,E1 -21638.464,E2 -21638.464} C_VEL
LIN {X 0,Y 204.988,Z 296.47,A -85,B 0,C 180,E1 -21641.129,E2 -21641.129} C_VEL
LIN {X 0,Y 209.607,Z 304.509,A -85,B 0,C 180,E1 -21643.178,E2 -21643.178} C_VEL
LIN {X 0,Y 213.948,Z 312.392,A -85,B 0,C 180,E1 -21644.925,E2 -21644.925} C_VEL
LIN {X 0,Y 216.647,Z 317.444,A -85,B 0,C 180,E1 -21645.951,E2 -21645.951} C_VEL
LIN {X 0,Y 222.544,Z 329.641,A -85,B 0,C 180,E1 -21648.089,E2 -21648.089} C_VEL
LIN {X 0,Y 226.285,Z 338.74,A -85,B 0,C 180,E1 -21649.409,E2 -21649.409} C_VEL
LIN {X 0,Y 227.648,Z 350.28,A -85,B 0,C 180,E1 -21650.219,E2 -21650.219} C_VEL
LIN {X 0,Y 227.764,Z 356.089,A -85,B 0,C 180,E1 -21650.489,E2 -21650.489} C_VEL
LIN {X 0,Y 225.226,Z 375.787,A -85,B 0,C 180,E1 -21650.738,E2 -21650.738} C_VEL
LIN {X 0,Y 225.176,Z 381.652,A -85,B 0,C 180,E1 -21650.974,E2 -21650.974} C_VEL
LIN {X 0,Y 225.376,Z 388.418,A -85,B 0,C 180,E1 -21651.303,E2 -21651.303} C_VEL
LIN {X 0,Y 223.932,Z 411.911,A -85,B 0,C 180,E1 -21652.038,E2 -21652.038} C_VEL
LIN {X 0,Y 222.146,Z 425.394,A -85,B 0,C 180,E1 -21652.735,E2 -21652.735} C_VEL
LIN {X 0,Y 219.802,Z 438.035,A -85,B 0,C 180,E1 -21653.735,E2 -21653.735} C_VEL
LIN {X 0,Y 216.558,Z 450.686,A -85,B 0,C 180,E1 -21655.111,E2 -21655.111} C_VEL
LIN {X 0,Y 212.846,Z 461.973,A -85,B 0,C 180,E1 -21656.705,E2 -21656.705} C_VEL
LIN {X 0,Y 209.042,Z 472.178,A -85,B 0,C 180,E1 -21658.593,E2 -21658.593} C_VEL
LIN {X 0,Y 205.274,Z 481.411,A -85,B 0,C 180,E1 -21660.798,E2 -21660.798} C_VEL
LIN {X 0,Y 201.288,Z 490.455,A -85,B 0,C 180,E1 -21663.566,E2 -21663.566} C_VEL
LIN {X 0,Y 197.925,Z 497.794,A -85,B 0,C 180,E1 -21666.455,E2 -21666.455} C_VEL
LIN {X 0,Y 194.927,Z 504.329,A -85,B 0,C 180,E1 -21669.817,E2 -21669.817} C_VEL
LIN {X 0,Y 192.995,Z 509.124,A -85,B 0,C 180,E1 -21673.062,E2 -21673.062} C_VEL
LIN {X 0,Y 191.654,Z 512.63,A -85,B 0,C 180,E1 -21676.21,E2 -21676.21} C_VEL
LIN {X 0,Y 191.012,Z 515.189,A -85,B 0,C 180,E1 -21679.398,E2 -21679.398} C_VEL
LIN {X 0,Y 191.179,Z 517.182,A -85,B 0,C 180,E1 -21683.668,E2 -21683.668} C_VEL
LIN {X 0,Y 191.458,Z 517.59,A -85,B 0,C 180,E1 -21685.789,E2 -21685.789} C_VEL
LIN {X 0,Y 191.843,Z 517.578,A -85,B 0,C 180,E1 -21687.9,E2 -21687.9} C_VEL
LIN {X 0,Y 192.013,Z 517.093,A -85,B 0,C 180,E1 -21689.999,E2 -21689.999} C_VEL
LIN {X 0,Y 191.917,Z 516.156,A -85,B 0,C 180,E1 -21692.098,E2 -21692.098} C_VEL
LIN {X 0,Y 191.583,Z 514.76,A -85,B 0,C 180,E1 -21694.206,E2 -21694.206} C_VEL
LIN {X 0,Y 191.212,Z 512.102,A -85,B 0,C 180,E1 -21697.077,E2 -21697.077} C_VEL
LIN {X 0,Y 191.184,Z 507.713,A -85,B 0,C 180,E1 -21700.59,E2 -21700.59} C_VEL
LIN {X 0,Y 191.874,Z 501.496,A -85,B 0,C 180,E1 -21704.313,E2 -21704.313} C_VEL
LIN {X 0,Y 193.048,Z 494.684,A -85,B 0,C 180,E1 -21707.477,E2 -21707.477} C_VEL
LIN {X 0,Y 195.115,Z 485.942,A -85,B 0,C 180,E1 -21710.685,E2 -21710.685} C_VEL
LIN {X 0,Y 197.115,Z 477.708,A -85,B 0,C 180,E1 -21713.09,E2 -21713.09} C_VEL
LIN {X 0,Y 199.339,Z 468.307,A -85,B 0,C 180,E1 -21715.306,E2 -21715.306} C_VEL
LIN {X 0,Y 202.01,Z 456.673,A -85,B 0,C 180,E1 -21717.448,E2 -21717.448} C_VEL
LIN {X 0,Y 204.275,Z 445.226,A -85,B 0,C 180,E1 -21719.074,E2 -21719.074} C_VEL
LIN {X 0,Y 206.121,Z 433.486,A -85,B 0,C 180,E1 -21720.333,E2 -21720.333} C_VEL
LIN {X 0,Y 207.665,Z 420.585,A -85,B 0,C 180,E1 -21721.305,E2 -21721.305} C_VEL
LIN {X 0,Y 208.478,Z 407.825,A -85,B 0,C 180,E1 -21721.935,E2 -21721.935} C_VEL
LIN {X 0,Y 209.416,Z 381.339,A -85,B 0,C 180,E1 -21722.819,E2 -21722.819} C_VEL
LIN {X 0,Y 206.813,Z 343.432,A -85,B 0,C 180,E1 -21724.697,E2 -21724.697} C_VEL
LIN {X 0,Y 204.325,Z 317.722,A -85,B 0,C 180,E1 -21726.143,E2 -21726.143} C_VEL
LIN {X 0,Y 198.857,Z 304.136,A -85,B 0,C 180,E1 -21727.688,E2 -21727.688} C_VEL
LIN {X 0,Y 197.457,Z 300.364,A -85,B 0,C 180,E1 -21728.21,E2 -21728.21} C_VEL
LIN {X 0,Y 194.925,Z 290.239,A -85,B 0,C 180,E1 -21732.345,E2 -21732.345} C_VEL
LIN {X 0,Y 192.5,Z 281.629,A -85,B 0,C 180,E1 -21736.267,E2 -21736.267} C_VEL
LIN {X 0,Y 192.537,Z 281.485,A -85,B 0,C 180,E1 -21741.645,E2 -21741.645} C_VEL
LIN {X 0,Y 192.588,Z 281.473,A -85,B 0,C 180,E1 -21746.813,E2 -21746.813} C_VEL
LIN {X 0,Y 192.613,Z 281.492,A -85,B 0,C 180,E1 -21751.684,E2 -21751.684} C_VEL
LIN {X 0,Y 192.663,Z 281.477,A -85,B 0,C 180,E1 -21756.343,E2 -21756.343} C_VEL
LIN {X 0,Y 192.687,Z 281.461,A -85,B 0,C 180,E1 -21761.491,E2 -21761.491} C_VEL
LIN {X 0,Y 192.727,Z 281.477,A -85,B 0,C 180,E1 -21765.211,E2 -21765.211} C_VEL
LIN {X 0,Y 192.938,Z 281.428,A -85,B 0,C 180,E1 -21769.567,E2 -21769.567} C_VEL
LIN {X 0,Y 192.957,Z 281.447,A -85,B 0,C 180,E1 -21773.727,E2 -21773.727} C_VEL
LIN {X 0,Y 193.222,Z 281.394,A -85,B 0,C 180,E1 -21777.916,E2 -21777.916} C_VEL
LIN {X 0,Y 193.404,Z 281.367,A -85,B 0,C 180,E1 -21780,E2 -21780} C_VEL
LIN {X 0,Y 192.918,Z 281.455,A -85,B 0,C 180,E1 -21784.179,E2 -21784.179} C_VEL
LIN {X 0,Y 193.01,Z 281.414,A -85,B 0,C 180,E1 -21788.375,E2 -21788.375} C_VEL
LIN {X 0,Y 192.781,Z 281.471,A -85,B 0,C 180,E1 -21792.635,E2 -21792.635} C_VEL
LIN {X 0,Y 192.709,Z 281.453,A -85,B 0,C 180,E1 -21796.964,E2 -21796.964} C_VEL
LIN {X 0,Y 192.573,Z 281.496,A -85,B 0,C 180,E1 -21801.405,E2 -21801.405} C_VEL
LIN {X 0,Y 192.612,Z 281.479,A -85,B 0,C 180,E1 -21804.194,E2 -21804.194} C_VEL
LIN {X 0,Y 192.589,Z 281.494,A -85,B 0,C 180,E1 -21808.863,E2 -21808.863} C_VEL
LIN {X 0,Y 192.59,Z 281.476,A -85,B 0,C 180,E1 -21813.188,E2 -21813.188} C_VEL
LIN {X 0,Y 192.537,Z 281.497,A -85,B 0,C 180,E1 -21818.356,E2 -21818.356} C_VEL
LIN {X 0,Y 192.479,Z 281.445,A -85,B 0,C 180,E1 -21823.094,E2 -21823.094} C_VEL
LIN {X 0,Y 192.482,Z 281.496,A -85,B 0,C 180,E1 -21826.908,E2 -21826.908} C_VEL
LIN {X 0,Y 192.539,Z 281.461,A -85,B 0,C 180,E1 -21831.647,E2 -21831.647} C_VEL
LIN {X 0,Y 192.594,Z 281.495,A -85,B 0,C 180,E1 -21836.815,E2 -21836.815} C_VEL
LIN {X 0,Y 192.594,Z 281.713,A -85,B 0,C 180,E1 -21839.601,E2 -21839.601} C_VEL
LIN {X 0,Y 192.856,Z 282.81,A -85,B 0,C 180,E1 -21839.952,E2 -21839.952} C_VEL
LIN {X 0,Y 194.462,Z 285.495,A -85,B 0,C 180,E1 -21840.427,E2 -21840.427} C_VEL
LIN {X 0,Y 201.117,Z 297.23,A -85,B 0,C 180,E1 -21842.232,E2 -21842.232} C_VEL
LIN {X 0,Y 208.694,Z 312.274,A -85,B 0,C 180,E1 -21844.175,E2 -21844.175} C_VEL
LIN {X 0,Y 211.755,Z 319.469,A -85,B 0,C 180,E1 -21844.955,E2 -21844.955} C_VEL
LIN {X 0,Y 210.228,Z 368.19,A -85,B 0,C 180,E1 -21846.641,E2 -21846.641} C_VEL
LIN {X 0,Y 209.586,Z 379.323,A -85,B 0,C 180,E1 -21847.309,E2 -21847.309} C_VEL
LIN {X 0,Y 208.4,Z 392.456,A -85,B 0,C 180,E1 -21848.486,E2 -21848.486} C_VEL
LIN {X 0,Y 206.869,Z 403.985,A -85,B 0,C 180,E1 -21849.882,E2 -21849.882} C_VEL
LIN {X 0,Y 205.03,Z 414.531,A -85,B 0,C 180,E1 -21851.515,E2 -21851.515} C_VEL
LIN {X 0,Y 202.938,Z 425.277,A -85,B 0,C 180,E1 -21853.659,E2 -21853.659} C_VEL
LIN {X 0,Y 200.99,Z 434.048,A -85,B 0,C 180,E1 -21855.833,E2 -21855.833} C_VEL
LIN {X 0,Y 198.637,Z 443.586,A -85,B 0,C 180,E1 -21858.78,E2 -21858.78} C_VEL
LIN {X 0,Y 196.637,Z 451.204,A -85,B 0,C 180,E1 -21861.782,E2 -21861.782} C_VEL
LIN {X 0,Y 195.095,Z 457.31,A -85,B 0,C 180,E1 -21864.834,E2 -21864.834} C_VEL
LIN {X 0,Y 193.881,Z 462.181,A -85,B 0,C 180,E1 -21867.924,E2 -21867.924} C_VEL
LIN {X 0,Y 192.947,Z 465.97,A -85,B 0,C 180,E1 -21871.044,E2 -21871.044} C_VEL
LIN {X 0,Y 192.525,Z 468.739,A -85,B 0,C 180,E1 -21874.188,E2 -21874.188} C_VEL
LIN {X 0,Y 192.504,Z 470.051,A -85,B 0,C 180,E1 -21876.289,E2 -21876.289} C_VEL
LIN {X 0,Y 192.718,Z 471.443,A -85,B 0,C 180,E1 -21880.053,E2 -21880.053} C_VEL
LIN {X 0,Y 193.1,Z 471.663,A -85,B 0,C 180,E1 -21882.614,E2 -21882.614} C_VEL
LIN {X 0,Y 194.403,Z 470.772,A -85,B 0,C 180,E1 -21886.811,E2 -21886.811} C_VEL
LIN {X 0,Y 195.305,Z 469.721,A -85,B 0,C 180,E1 -21888.897,E2 -21888.897} C_VEL
LIN {X 0,Y 197.172,Z 467.266,A -85,B 0,C 180,E1 -21892.065,E2 -21892.065} C_VEL
LIN {X 0,Y 199.268,Z 463.966,A -85,B 0,C 180,E1 -21895.039,E2 -21895.039} C_VEL
LIN {X 0,Y 201.847,Z 459.464,A -85,B 0,C 180,E1 -21898.038,E2 -21898.038} C_VEL
LIN {X 0,Y 205.448,Z 452.579,A -85,B 0,C 180,E1 -21901.445,E2 -21901.445} C_VEL
LIN {X 0,Y 208.956,Z 445.068,A -85,B 0,C 180,E1 -21904.289,E2 -21904.289} C_VEL
